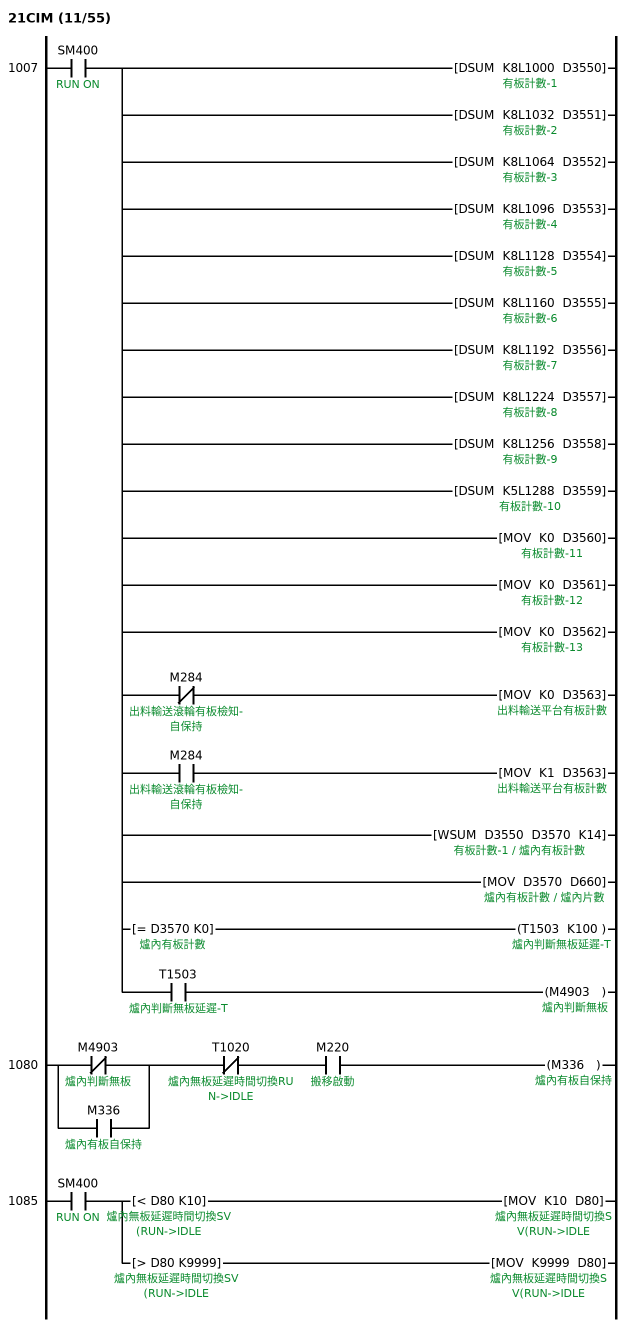
[picture p120: ladder of 21CIM, rungs at steps 1007 to 1085]
1007  LD      SM400  ; RUN ON
      DSUM    K8L1000 D3550  ; 上板記憶 / 有板計數-1
      DSUM    K8L1032 D3551  ; 上板記憶 / 有板計數-2
      DSUM    K8L1064 D3552  ; 上板記憶 / 有板計數-3
      DSUM    K8L1096 D3553  ; 上板記憶 / 有板計數-4
      DSUM    K8L1128 D3554  ; 上板記憶 / 有板計數-5
      DSUM    K8L1160 D3555  ; 上板記憶 / 有板計數-6
      DSUM    K8L1192 D3556  ; 上板記憶 / 有板計數-7
      DSUM    K8L1224 D3557  ; 上板記憶 / 有板計數-8
      DSUM    K8L1256 D3558  ; 上板記憶 / 有板計數-9
      DSUM    K5L1288 D3559  ; 上板記憶 / 有板計數-10
      MOV     K0 D3560  ; 有板計數-11
      MOV     K0 D3561  ; 有板計數-12
      MOV     K0 D3562  ; 有板計數-13
      MPS
      ANI     M284  ; 出料輸送滾輪有板檢知-自保持
      MOV     K0 D3563  ; 出料輸送平台有板計數
      MRD
      AND     M284  ; 出料輸送滾輪有板檢知-自保持
      MOV     K1 D3563
      MPP
      WSUM    D3550 D3570 K14  ; 爐內有板計數
      MOV     D3570 D660  ; 爐內片數
      MPS
      AND=    D3570 K0  ; 爐內有板計數
      OUT     T1503 K100  ; 爐內判斷無板延遲-T
      MPP
      AND     T1503  ; 爐內判斷無板延遲-T
      OUT     M4903  ; 爐內判斷無板
1080  LDI     M4903  ; 爐內判斷無板
      OR      M336  ; 爐內有板自保持
      ANI     T1020  ; 爐內無板延遲時間切換RUN->IDLE
      AND     M220  ; 搬移啟動
      OUT     M336  ; 爐內有板自保持
1085  LD      SM400  ; RUN ON
      MPS
      AND<    D80 K10  ; 爐內無板延遲時間切換SV(RUN->IDLE
      MOV     K10 D80
      MPP
      AND>    D80 K9999  ; 爐內無板延遲時間切換SV(RUN->IDLE
      MOV     K9999 D80
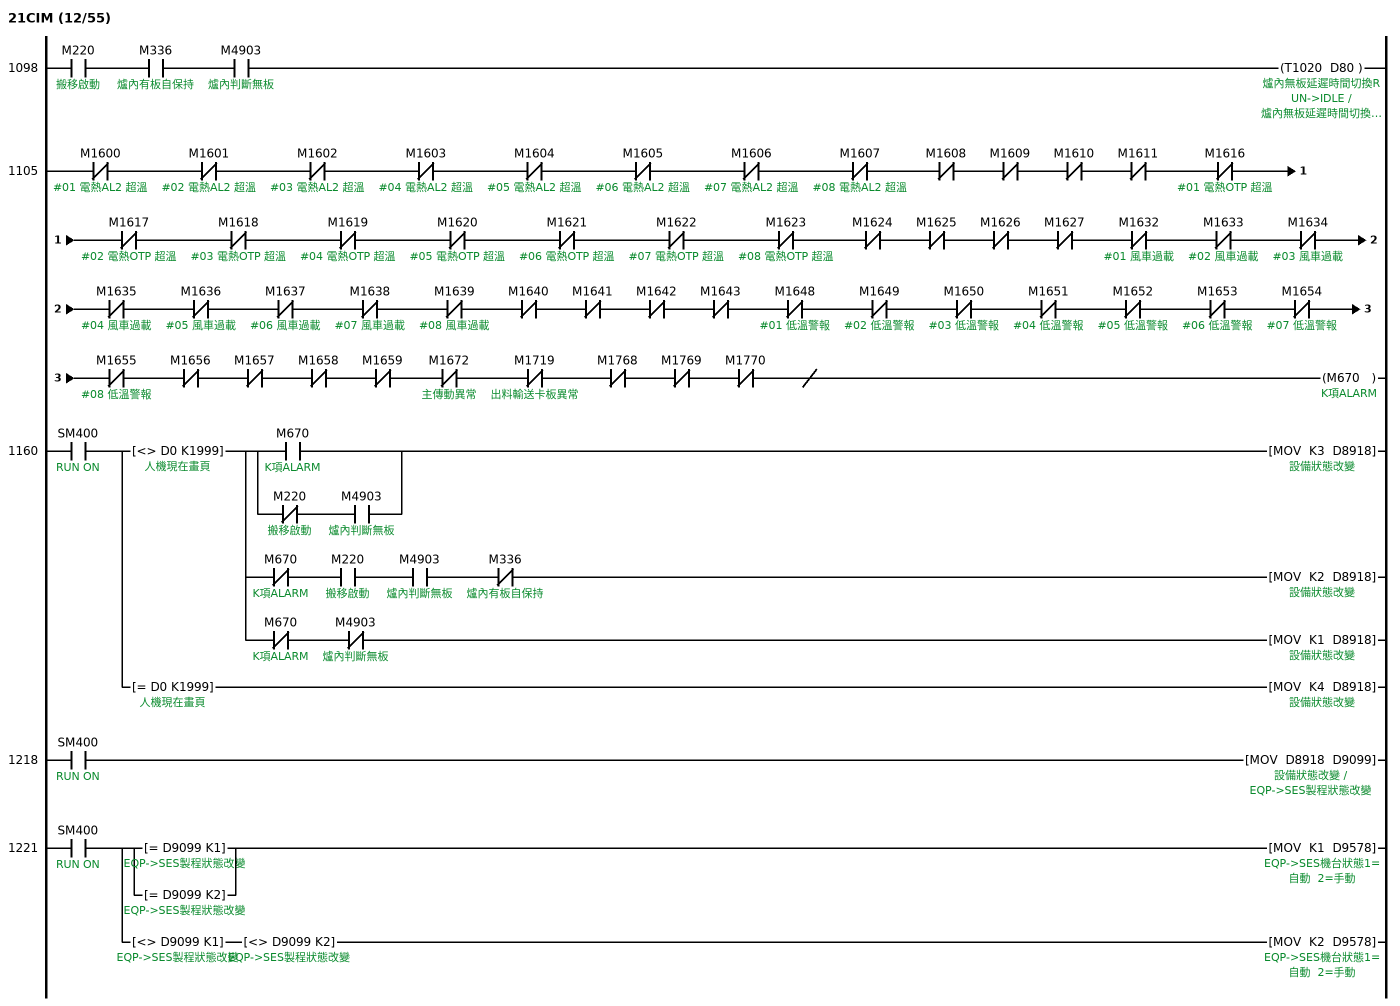
1098  LD      M220  ; 搬移啟動
      AND     M336  ; 爐內有板自保持
      AND     M4903  ; 爐內判斷無板
      OUT     T1020 D80  ; 爐內無板延遲時間切換RUN->IDLE / 爐內無板延遲時間切換SV(RUN->IDLE
1105  LDI     M1600  ; #01 電熱AL2 超溫
      ANI     M1601  ; #02 電熱AL2 超溫
      ANI     M1602  ; #03 電熱AL2 超溫
      ANI     M1603  ; #04 電熱AL2 超溫
      ANI     M1604  ; #05 電熱AL2 超溫
      ANI     M1605  ; #06 電熱AL2 超溫
      ANI     M1606  ; #07 電熱AL2 超溫
      ANI     M1607  ; #08 電熱AL2 超溫
      ANI     M1608
      ANI     M1609
      ANI     M1610
      ANI     M1611
      ANI     M1616  ; #01 電熱OTP 超溫
      ANI     M1617  ; #02 電熱OTP 超溫
      ANI     M1618  ; #03 電熱OTP 超溫
      ANI     M1619  ; #04 電熱OTP 超溫
      ANI     M1620  ; #05 電熱OTP 超溫
      ANI     M1621  ; #06 電熱OTP 超溫
      ANI     M1622  ; #07 電熱OTP 超溫
      ANI     M1623  ; #08 電熱OTP 超溫
      ANI     M1624
      ANI     M1625
      ANI     M1626
      ANI     M1627
      ANI     M1632  ; #01 風車過載
      ANI     M1633  ; #02 風車過載
      ANI     M1634  ; #03 風車過載
      ANI     M1635  ; #04 風車過載
      ANI     M1636  ; #05 風車過載
      ANI     M1637  ; #06 風車過載
      ANI     M1638  ; #07 風車過載
      ANI     M1639  ; #08 風車過載
      ANI     M1640
      ANI     M1641
      ANI     M1642
      ANI     M1643
      ANI     M1648  ; #01 低溫警報
      ANI     M1649  ; #02 低溫警報
      ANI     M1650  ; #03 低溫警報
      ANI     M1651  ; #04 低溫警報
      ANI     M1652  ; #05 低溫警報
      ANI     M1653  ; #06 低溫警報
      ANI     M1654  ; #07 低溫警報
      ANI     M1655  ; #08 低溫警報
      ANI     M1656
      ANI     M1657
      ANI     M1658
      ANI     M1659
      ANI     M1672  ; 主傳動異常
      ANI     M1719  ; 出料輸送卡板異常
      ANI     M1768
      ANI     M1769
      ANI     M1770
      INV
      OUT     M670  ; K項ALARM
1160  LD      SM400  ; RUN ON
      MPS
      AND<>   D0 K1999  ; 人機現在畫頁
      MPS
      LD      M670  ; K項ALARM
      LDI     M220  ; 搬移啟動
      AND     M4903  ; 爐內判斷無板
      ORB
      ANB
      MOV     K3 D8918  ; 設備狀態改變
        [note] State=DOWN
      MRD
      ANI     M670  ; K項ALARM
      AND     M220  ; 搬移啟動
      AND     M4903  ; 爐內判斷無板
      ANI     M336  ; 爐內有板自保持
      MOV     K2 D8918
        [note] State=IDLE
      MPP
      ANI     M670  ; K項ALARM
      ANI     M4903  ; 爐內判斷無板
      MOV     K1 D8918
        [note] State=RUN
      MPP
      AND=    D0 K1999  ; 人機現在畫頁
      MOV     K4 D8918
        [note] State=PM
1218  LD      SM400  ; RUN ON
      MOV     D8918 D9099  ; EQP->SES製程狀態改變
1221  LD      SM400  ; RUN ON
      MPS
      LD=     D9099 K1  ; EQP->SES製程狀態改變
      OR=     D9099 K2  ; EQP->SES製程狀態改變
      ANB
      MOV     K1 D9578  ; EQP->SES機台狀態1=自動  2=手動
      MPP
      AND<>   D9099 K1  ; EQP->SES製程狀態改變
      AND<>   D9099 K2  ; EQP->SES製程狀態改變
      MOV     K2 D9578
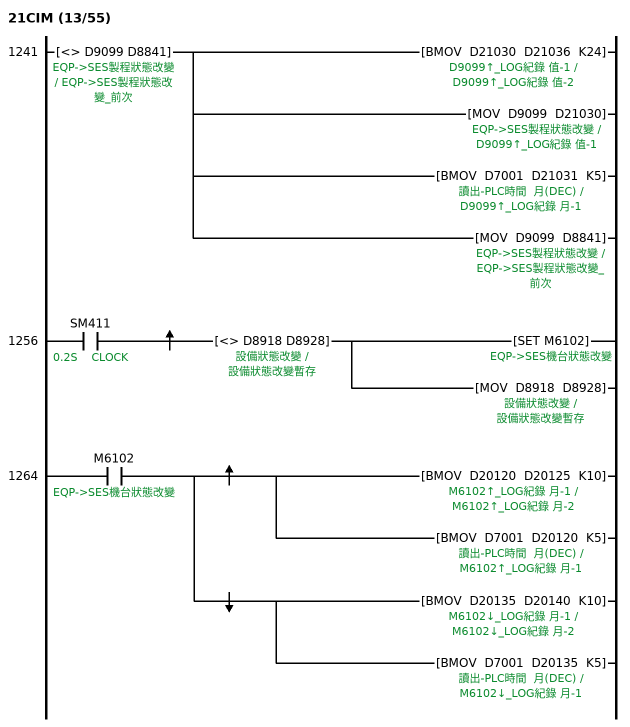
1241  LD<>    D9099 D8841  ; EQP->SES製程狀態改變 / EQP->SES製程狀態改變_前次
      BMOV    D21030 D21036 K24  ; D9099↑_LOG紀錄 值-1 / D9099↑_LOG紀錄 值-2
      MOV     D9099 D21030
      BMOV    D7001 D21031 K5  ; D9099↑_LOG紀錄 月-1
      MOV     D9099 D8841
1256  LD      SM411  ; 0.2S    CLOCK
      MEP
      AND<>   D8918 D8928  ; 設備狀態改變 / 設備狀態改變暫存
      SET     M6102  ; EQP->SES機台狀態改變
      MOV     D8918 D8928
1264  LD      M6102  ; EQP->SES機台狀態改變
      MPS
      MEP
      BMOV    D20120 D20125 K10  ; M6102↑_LOG紀錄 月-1 / M6102↑_LOG紀錄 月-2
      BMOV    D7001 D20120 K5
      MPP
      MEF
      BMOV    D20135 D20140 K10  ; M6102↓_LOG紀錄 月-1 / M6102↓_LOG紀錄 月-2
      BMOV    D7001 D20135 K5
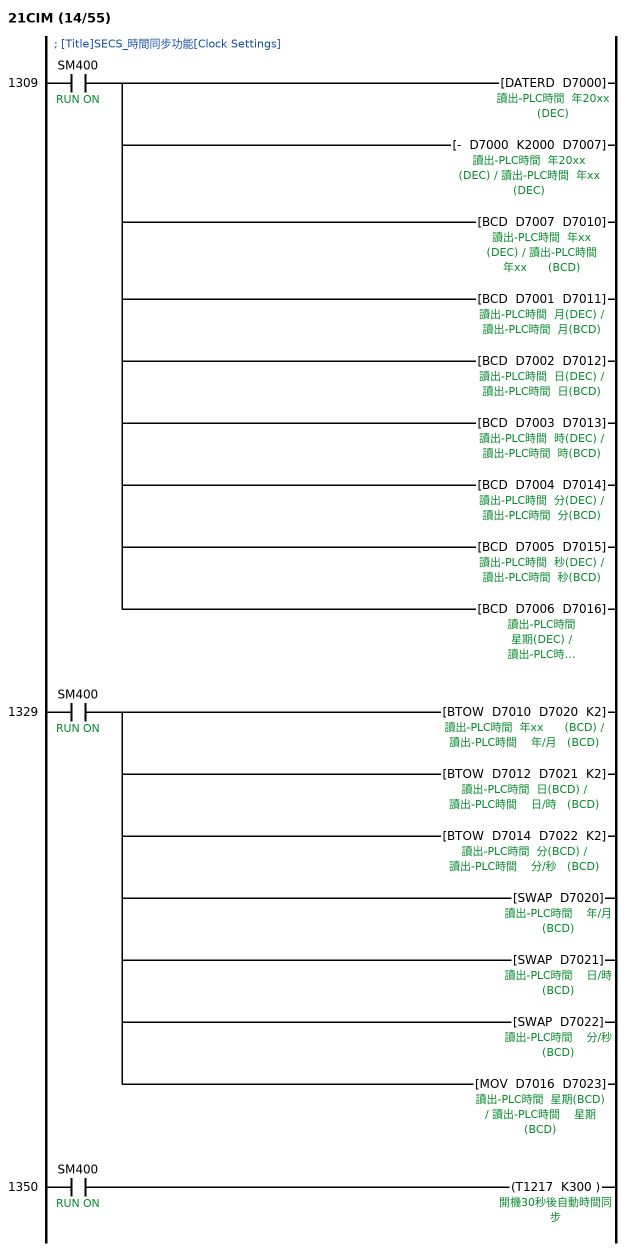
; [Title]SECS_時間同步功能[Clock Settings]
1309  LD      SM400  ; RUN ON
      DATERD  D7000  ; 讀出-PLC時間  年20xx    (DEC)
      -       D7000 K2000 D7007  ; 讀出-PLC時間  年xx      (DEC)
      BCD     D7007 D7010  ; 讀出-PLC時間  年xx      (BCD)
      BCD     D7001 D7011  ; 讀出-PLC時間  月(BCD)
      BCD     D7002 D7012  ; 讀出-PLC時間  日(DEC) / 讀出-PLC時間  日(BCD)
      BCD     D7003 D7013  ; 讀出-PLC時間  時(DEC) / 讀出-PLC時間  時(BCD)
      BCD     D7004 D7014  ; 讀出-PLC時間  分(DEC) / 讀出-PLC時間  分(BCD)
      BCD     D7005 D7015  ; 讀出-PLC時間  秒(DEC) / 讀出-PLC時間  秒(BCD)
      BCD     D7006 D7016  ; 讀出-PLC時間  星期(DEC) / 讀出-PLC時間  星期(BCD)
1329  LD      SM400  ; RUN ON
      BTOW    D7010 D7020 K2  ; 讀出-PLC時間    年/月   (BCD)
      BTOW    D7012 D7021 K2  ; 讀出-PLC時間    日/時   (BCD)
      BTOW    D7014 D7022 K2  ; 讀出-PLC時間    分/秒   (BCD)
      SWAP    D7020
      SWAP    D7021
      SWAP    D7022
      MOV     D7016 D7023  ; 讀出-PLC時間    星期    (BCD)
1350  LD      SM400  ; RUN ON
      OUT     T1217 K300  ; 開機30秒後自動時間同步
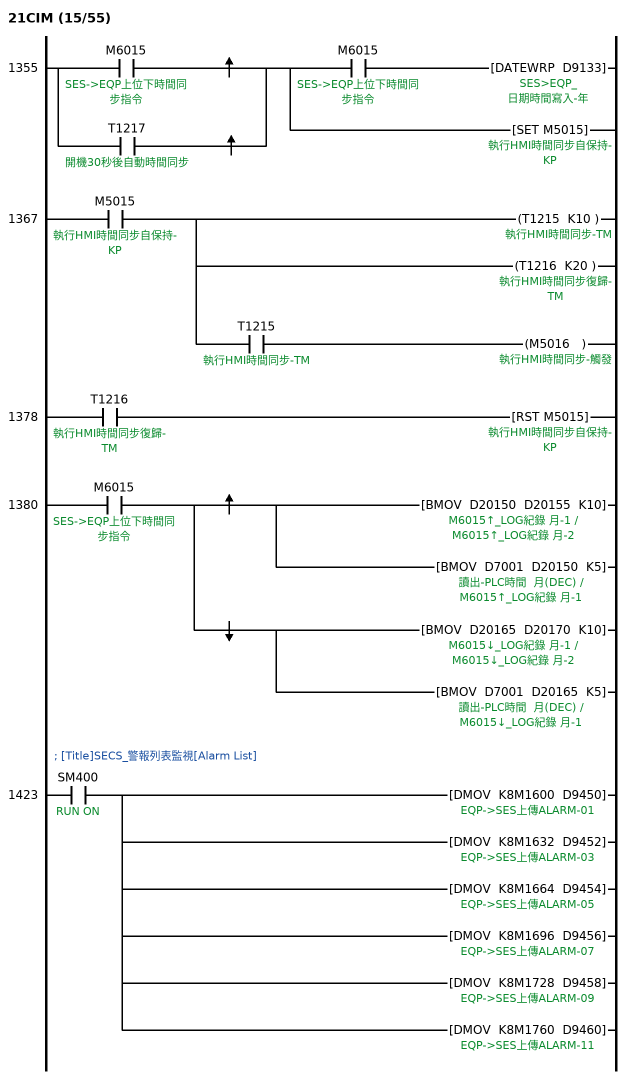
1355  LD      M6015  ; SES->EQP上位下時間同步指令
      MEP
      LD      T1217  ; 開機30秒後自動時間同步
      MEP
      ORB
      MPS
      AND     M6015  ; SES->EQP上位下時間同步指令
      DATEWRP D9133  ; SES>EQP_日期時間寫入-年
      MPP
      SET     M5015  ; 執行HMI時間同步自保持-KP
1367  LD      M5015  ; 執行HMI時間同步自保持-KP
      OUT     T1215 K10  ; 執行HMI時間同步-TM
      OUT     T1216 K20  ; 執行HMI時間同步復歸-TM
      AND     T1215  ; 執行HMI時間同步-TM
      OUT     M5016  ; 執行HMI時間同步-觸發
1378  LD      T1216  ; 執行HMI時間同步復歸-TM
      RST     M5015  ; 執行HMI時間同步自保持-KP
1380  LD      M6015  ; SES->EQP上位下時間同步指令
      MPS
      MEP
      BMOV    D20150 D20155 K10  ; M6015↑_LOG紀錄 月-1 / M6015↑_LOG紀錄 月-2
      BMOV    D7001 D20150 K5
      MPP
      MEF
      BMOV    D20165 D20170 K10  ; M6015↓_LOG紀錄 月-1 / M6015↓_LOG紀錄 月-2
      BMOV    D7001 D20165 K5
; [Title]SECS_警報列表監視[Alarm List]
1423  LD      SM400  ; RUN ON
      DMOV    K8M1600 D9450  ; EQP->SES上傳ALARM-01
      DMOV    K8M1632 D9452  ; EQP->SES上傳ALARM-03
      DMOV    K8M1664 D9454  ; EQP->SES上傳ALARM-05
      DMOV    K8M1696 D9456  ; EQP->SES上傳ALARM-07
      DMOV    K8M1728 D9458  ; EQP->SES上傳ALARM-09
      DMOV    K8M1760 D9460  ; EQP->SES上傳ALARM-11
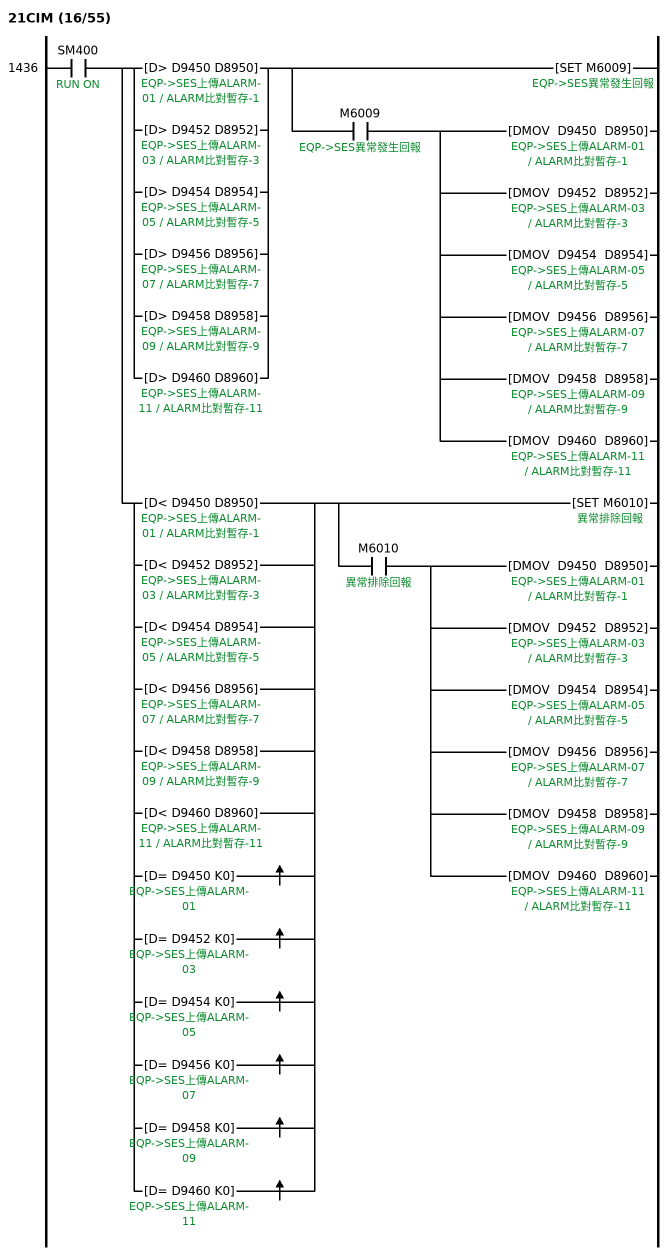
1436  LD      SM400  ; RUN ON
      MPS
      LDD>    D9450 D8950  ; EQP->SES上傳ALARM-01 / ALARM比對暫存-1
      ORD>    D9452 D8952  ; EQP->SES上傳ALARM-03 / ALARM比對暫存-3
      ORD>    D9454 D8954  ; EQP->SES上傳ALARM-05 / ALARM比對暫存-5
      ORD>    D9456 D8956  ; EQP->SES上傳ALARM-07 / ALARM比對暫存-7
      ORD>    D9458 D8958  ; EQP->SES上傳ALARM-09 / ALARM比對暫存-9
      ORD>    D9460 D8960  ; EQP->SES上傳ALARM-11 / ALARM比對暫存-11
      ANB
      SET     M6009  ; EQP->SES異常發生回報
      AND     M6009  ; EQP->SES異常發生回報
      DMOV    D9450 D8950
      DMOV    D9452 D8952
      DMOV    D9454 D8954
      DMOV    D9456 D8956
      DMOV    D9458 D8958
      DMOV    D9460 D8960
      MPP
      LDD<    D9450 D8950  ; EQP->SES上傳ALARM-01 / ALARM比對暫存-1
      ORD<    D9452 D8952  ; EQP->SES上傳ALARM-03 / ALARM比對暫存-3
      ORD<    D9454 D8954  ; EQP->SES上傳ALARM-05 / ALARM比對暫存-5
      ORD<    D9456 D8956  ; EQP->SES上傳ALARM-07 / ALARM比對暫存-7
      ORD<    D9458 D8958  ; EQP->SES上傳ALARM-09 / ALARM比對暫存-9
      ORD<    D9460 D8960  ; EQP->SES上傳ALARM-11 / ALARM比對暫存-11
      LDD=    D9450 K0  ; EQP->SES上傳ALARM-01
      MEP
      ORB
      LDD=    D9452 K0  ; EQP->SES上傳ALARM-03
      MEP
      ORB
      LDD=    D9454 K0  ; EQP->SES上傳ALARM-05
      MEP
      ORB
      LDD=    D9456 K0  ; EQP->SES上傳ALARM-07
      MEP
      ORB
      LDD=    D9458 K0  ; EQP->SES上傳ALARM-09
      MEP
      ORB
      LDD=    D9460 K0  ; EQP->SES上傳ALARM-11
      MEP
      ORB
      ANB
      SET     M6010  ; 異常排除回報
      AND     M6010  ; 異常排除回報
      DMOV    D9450 D8950
      DMOV    D9452 D8952
      DMOV    D9454 D8954
      DMOV    D9456 D8956
      DMOV    D9458 D8958
      DMOV    D9460 D8960
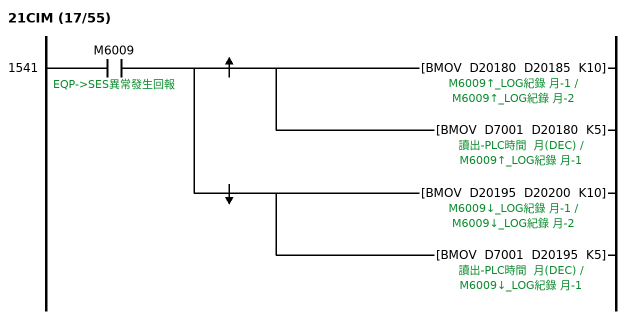
1541  LD      M6009  ; EQP->SES異常發生回報
      MPS
      MEP
      BMOV    D20180 D20185 K10  ; M6009↑_LOG紀錄 月-1 / M6009↑_LOG紀錄 月-2
      BMOV    D7001 D20180 K5
      MPP
      MEF
      BMOV    D20195 D20200 K10  ; M6009↓_LOG紀錄 月-1 / M6009↓_LOG紀錄 月-2
      BMOV    D7001 D20195 K5
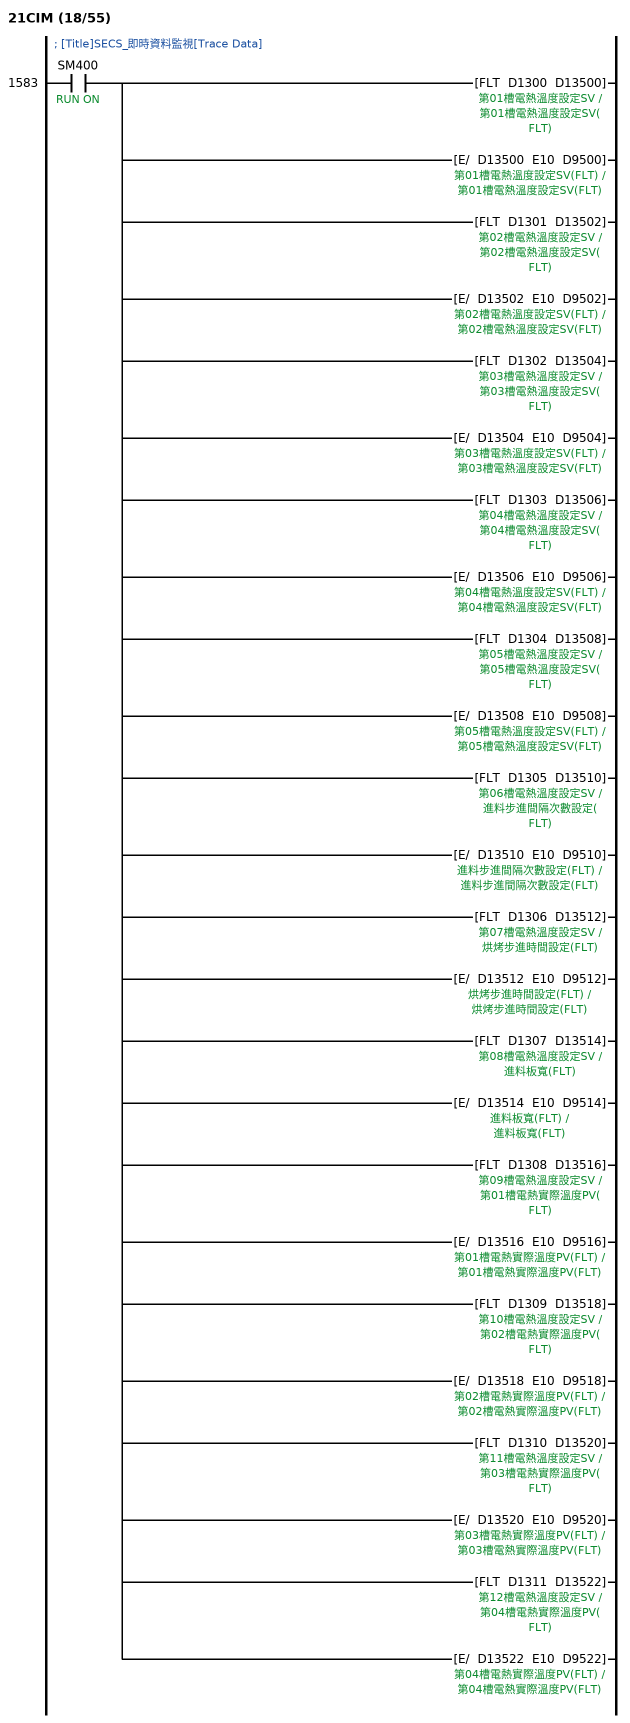
; [Title]SECS_即時資料監視[Trace Data]
1583  LD      SM400  ; RUN ON
      FLT     D1300 D13500  ; 第01槽電熱溫度設定SV(FLT)
      E/      D13500 E10 D9500  ; 第01槽電熱溫度設定SV(FLT)
      FLT     D1301 D13502  ; 第02槽電熱溫度設定SV / 第02槽電熱溫度設定SV(FLT)
      E/      D13502 E10 D9502  ; 第02槽電熱溫度設定SV(FLT)
      FLT     D1302 D13504  ; 第03槽電熱溫度設定SV / 第03槽電熱溫度設定SV(FLT)
      E/      D13504 E10 D9504  ; 第03槽電熱溫度設定SV(FLT)
      FLT     D1303 D13506  ; 第04槽電熱溫度設定SV / 第04槽電熱溫度設定SV(FLT)
      E/      D13506 E10 D9506  ; 第04槽電熱溫度設定SV(FLT)
      FLT     D1304 D13508  ; 第05槽電熱溫度設定SV / 第05槽電熱溫度設定SV(FLT)
      E/      D13508 E10 D9508  ; 第05槽電熱溫度設定SV(FLT)
      FLT     D1305 D13510  ; 第06槽電熱溫度設定SV / 進料步進間隔次數設定(FLT)
      E/      D13510 E10 D9510  ; 進料步進間隔次數設定(FLT)
      FLT     D1306 D13512  ; 第07槽電熱溫度設定SV / 烘烤步進時間設定(FLT)
      E/      D13512 E10 D9512  ; 烘烤步進時間設定(FLT)
      FLT     D1307 D13514  ; 第08槽電熱溫度設定SV / 進料板寬(FLT)
      E/      D13514 E10 D9514  ; 進料板寬(FLT)
      FLT     D1308 D13516  ; 第09槽電熱溫度設定SV / 第01槽電熱實際溫度PV(FLT)
      E/      D13516 E10 D9516  ; 第01槽電熱實際溫度PV(FLT)
      FLT     D1309 D13518  ; 第10槽電熱溫度設定SV / 第02槽電熱實際溫度PV(FLT)
      E/      D13518 E10 D9518  ; 第02槽電熱實際溫度PV(FLT)
      FLT     D1310 D13520  ; 第11槽電熱溫度設定SV / 第03槽電熱實際溫度PV(FLT)
      E/      D13520 E10 D9520  ; 第03槽電熱實際溫度PV(FLT)
      FLT     D1311 D13522  ; 第12槽電熱溫度設定SV / 第04槽電熱實際溫度PV(FLT)
      E/      D13522 E10 D9522  ; 第04槽電熱實際溫度PV(FLT)
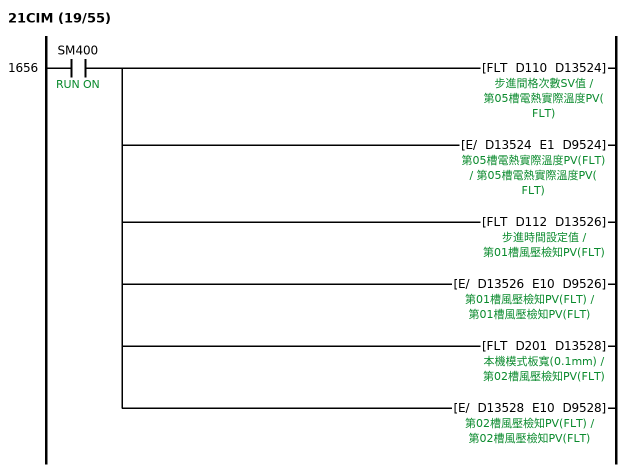
1656  LD      SM400  ; RUN ON
      FLT     D110 D13524  ; 第05槽電熱實際溫度PV(FLT)
      E/      D13524 E1 D9524  ; 第05槽電熱實際溫度PV(FLT)
      FLT     D112 D13526  ; 第01槽風壓檢知PV(FLT)
      E/      D13526 E10 D9526  ; 第01槽風壓檢知PV(FLT)
      FLT     D201 D13528  ; 第02槽風壓檢知PV(FLT)
      E/      D13528 E10 D9528  ; 第02槽風壓檢知PV(FLT)
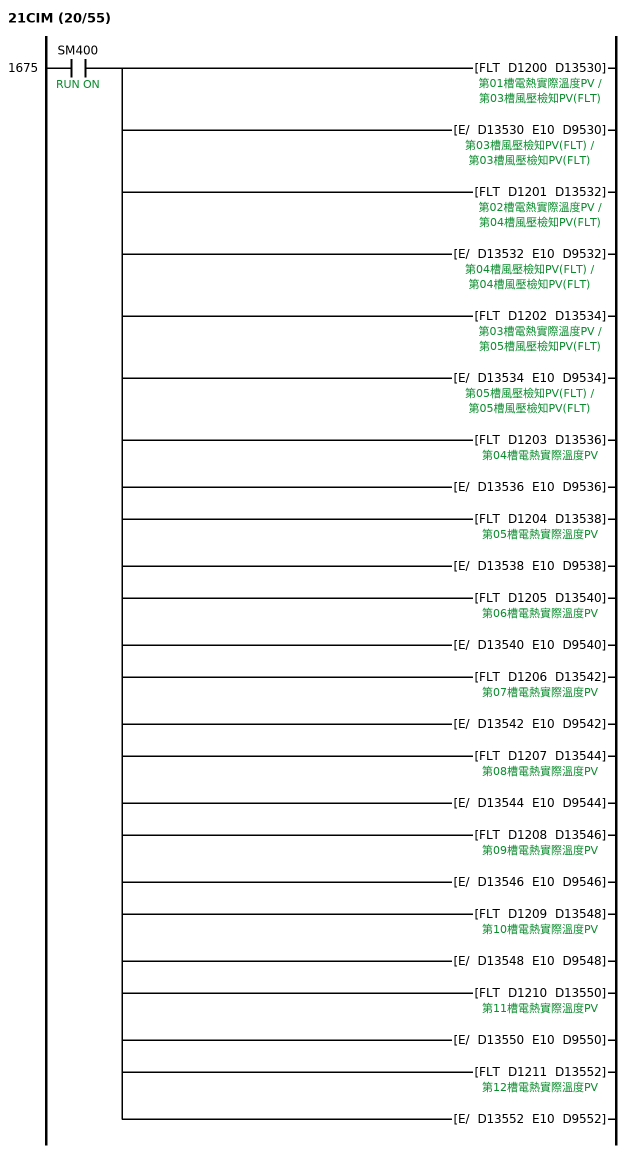
1675  LD      SM400  ; RUN ON
      FLT     D1200 D13530  ; 第03槽風壓檢知PV(FLT)
      E/      D13530 E10 D9530  ; 第03槽風壓檢知PV(FLT)
      FLT     D1201 D13532  ; 第02槽電熱實際溫度PV / 第04槽風壓檢知PV(FLT)
      E/      D13532 E10 D9532  ; 第04槽風壓檢知PV(FLT)
      FLT     D1202 D13534  ; 第03槽電熱實際溫度PV / 第05槽風壓檢知PV(FLT)
      E/      D13534 E10 D9534  ; 第05槽風壓檢知PV(FLT)
      FLT     D1203 D13536  ; 第04槽電熱實際溫度PV
      E/      D13536 E10 D9536
      FLT     D1204 D13538  ; 第05槽電熱實際溫度PV
      E/      D13538 E10 D9538
      FLT     D1205 D13540  ; 第06槽電熱實際溫度PV
      E/      D13540 E10 D9540
      FLT     D1206 D13542  ; 第07槽電熱實際溫度PV
      E/      D13542 E10 D9542
      FLT     D1207 D13544  ; 第08槽電熱實際溫度PV
      E/      D13544 E10 D9544
      FLT     D1208 D13546  ; 第09槽電熱實際溫度PV
      E/      D13546 E10 D9546
      FLT     D1209 D13548  ; 第10槽電熱實際溫度PV
      E/      D13548 E10 D9548
      FLT     D1210 D13550  ; 第11槽電熱實際溫度PV
      E/      D13550 E10 D9550
      FLT     D1211 D13552
      E/      D13552 E10 D9552
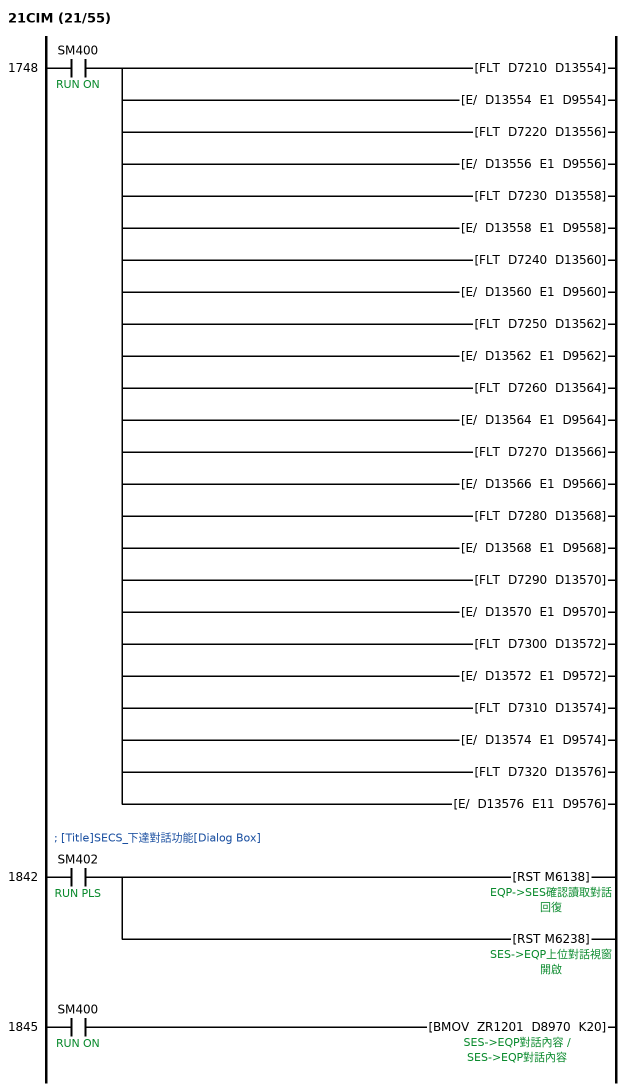
1748  LD      SM400  ; RUN ON
      FLT     D7210 D13554
      E/      D13554 E1 D9554
      FLT     D7220 D13556
      E/      D13556 E1 D9556
      FLT     D7230 D13558
      E/      D13558 E1 D9558
      FLT     D7240 D13560
      E/      D13560 E1 D9560
      FLT     D7250 D13562
      E/      D13562 E1 D9562
      FLT     D7260 D13564
      E/      D13564 E1 D9564
      FLT     D7270 D13566
      E/      D13566 E1 D9566
      FLT     D7280 D13568
      E/      D13568 E1 D9568
      FLT     D7290 D13570
      E/      D13570 E1 D9570
      FLT     D7300 D13572
      E/      D13572 E1 D9572
      FLT     D7310 D13574
      E/      D13574 E1 D9574
      FLT     D7320 D13576
      E/      D13576 E11 D9576
; [Title]SECS_下達對話功能[Dialog Box]
1842  LD      SM402  ; RUN PLS
      RST     M6138  ; EQP->SES確認讀取對話回復
      RST     M6238  ; SES->EQP上位對話視窗開啟
1845  LD      SM400  ; RUN ON
      BMOV    ZR1201 D8970 K20  ; SES->EQP對話內容 / SES->EQP對話內容
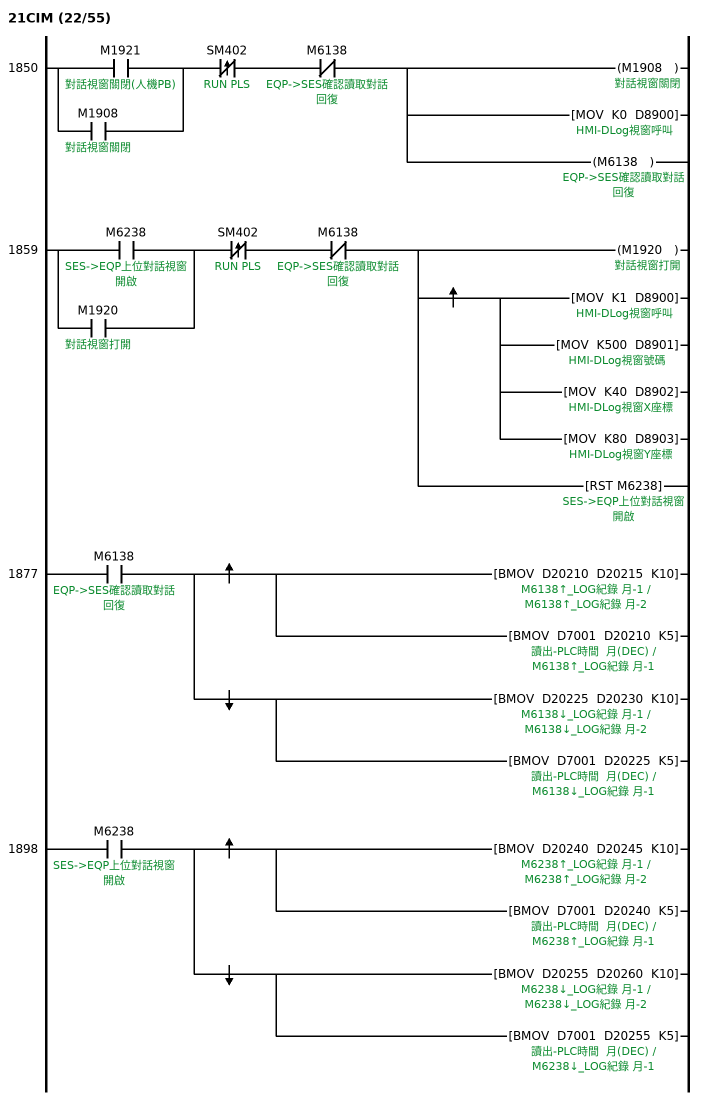
1850  LD      M1921  ; 對話視窗關閉(人機PB)
      OR      M1908  ; 對話視窗關閉
      ANDPI   SM402  ; RUN PLS
      ANI     M6138  ; EQP->SES確認讀取對話回復
      OUT     M1908  ; 對話視窗關閉
      MOV     K0 D8900  ; HMI-DLog視窗呼叫
      OUT     M6138  ; EQP->SES確認讀取對話回復
1859  LD      M6238  ; SES->EQP上位對話視窗開啟
      OR      M1920  ; 對話視窗打開
      ANDPI   SM402  ; RUN PLS
      ANI     M6138  ; EQP->SES確認讀取對話回復
      OUT     M1920  ; 對話視窗打開
      MPS
      MEP
      MOV     K1 D8900
      MOV     K500 D8901  ; HMI-DLog視窗號碼
      MOV     K40 D8902  ; HMI-DLog視窗X座標
      MOV     K80 D8903  ; HMI-DLog視窗Y座標
      MPP
      RST     M6238  ; SES->EQP上位對話視窗開啟
1877  LD      M6138  ; EQP->SES確認讀取對話回復
      MPS
      MEP
      BMOV    D20210 D20215 K10  ; M6138↑_LOG紀錄 月-1 / M6138↑_LOG紀錄 月-2
      BMOV    D7001 D20210 K5
      MPP
      MEF
      BMOV    D20225 D20230 K10  ; M6138↓_LOG紀錄 月-1 / M6138↓_LOG紀錄 月-2
      BMOV    D7001 D20225 K5
1898  LD      M6238  ; SES->EQP上位對話視窗開啟
      MPS
      MEP
      BMOV    D20240 D20245 K10  ; M6238↑_LOG紀錄 月-1 / M6238↑_LOG紀錄 月-2
      BMOV    D7001 D20240 K5
      MPP
      MEF
      BMOV    D20255 D20260 K10  ; M6238↓_LOG紀錄 月-1 / M6238↓_LOG紀錄 月-2
      BMOV    D7001 D20255 K5
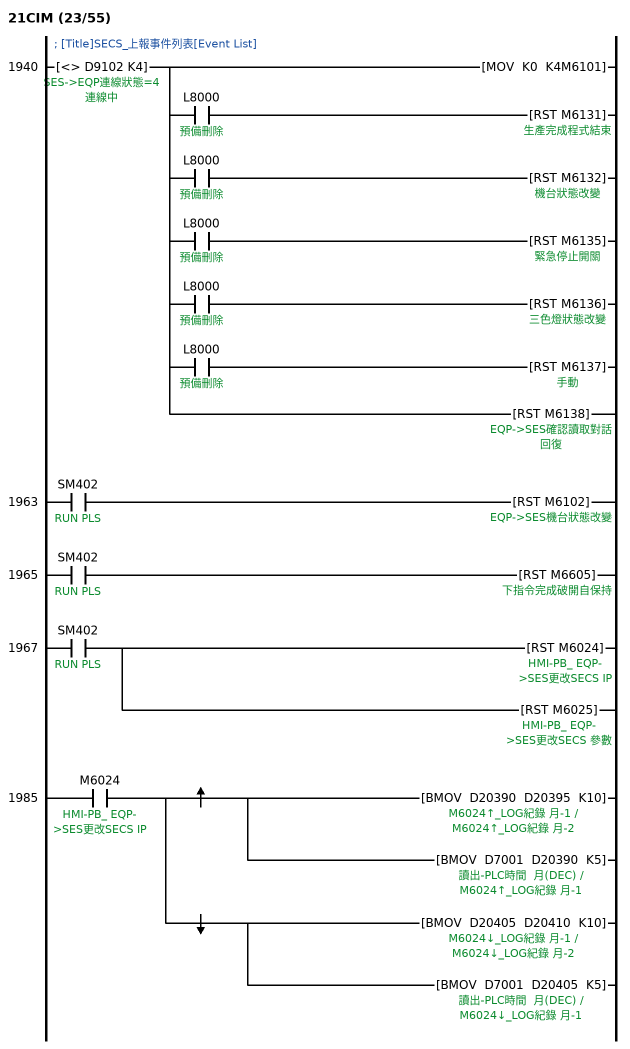
; [Title]SECS_上報事件列表[Event List]
1940  LD<>    D9102 K4  ; SES->EQP連線狀態=4      連線中
      MOV     K0 K4M6101
      MPS
      AND     L8000  ; 預備刪除
      RST     M6131  ; 生產完成程式結束
      MRD
      AND     L8000  ; 預備刪除
      RST     M6132  ; 機台狀態改變
      MRD
      AND     L8000  ; 預備刪除
      RST     M6135  ; 緊急停止開關
      MRD
      AND     L8000  ; 預備刪除
      RST     M6136  ; 三色燈狀態改變
      MRD
      AND     L8000  ; 預備刪除
      RST     M6137  ; 手動
      MPP
      RST     M6138  ; EQP->SES確認讀取對話回復
1963  LD      SM402  ; RUN PLS
      RST     M6102  ; EQP->SES機台狀態改變
1965  LD      SM402  ; RUN PLS
      RST     M6605  ; 下指令完成破開自保持
1967  LD      SM402  ; RUN PLS
      RST     M6024  ; HMI-PB_ EQP->SES更改SECS IP
        [note] HMI上變更C語言模組網路設定
      RST     M6025  ; HMI-PB_ EQP->SES更改SECS 參數
1985  LD      M6024  ; HMI-PB_ EQP->SES更改SECS IP
      MPS
      MEP
      BMOV    D20390 D20395 K10  ; M6024↑_LOG紀錄 月-1 / M6024↑_LOG紀錄 月-2
      BMOV    D7001 D20390 K5
      MPP
      MEF
      BMOV    D20405 D20410 K10  ; M6024↓_LOG紀錄 月-1 / M6024↓_LOG紀錄 月-2
      BMOV    D7001 D20405 K5
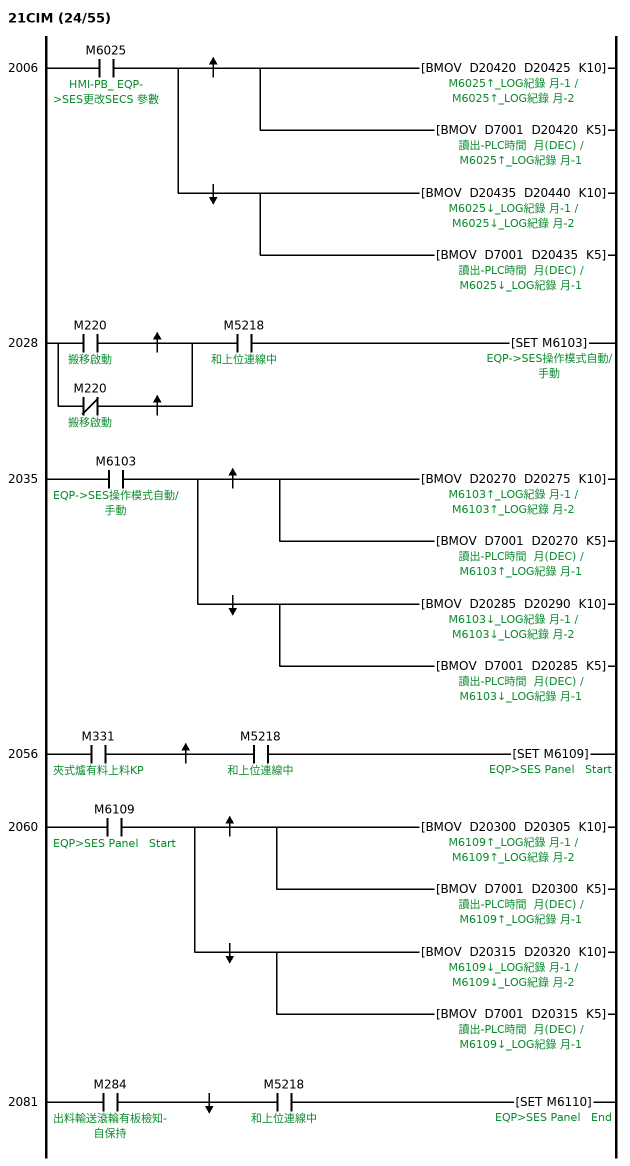
2006  LD      M6025  ; HMI-PB_ EQP->SES更改SECS 參數
      MPS
      MEP
      BMOV    D20420 D20425 K10  ; M6025↑_LOG紀錄 月-1 / M6025↑_LOG紀錄 月-2
      BMOV    D7001 D20420 K5
      MPP
      MEF
      BMOV    D20435 D20440 K10  ; M6025↓_LOG紀錄 月-1 / M6025↓_LOG紀錄 月-2
      BMOV    D7001 D20435 K5
2028  LD      M220  ; 搬移啟動
      MEP
      LDI     M220  ; 搬移啟動
      MEP
      ORB
      AND     M5218  ; 和上位連線中
      SET     M6103  ; EQP->SES操作模式自動/手動
2035  LD      M6103  ; EQP->SES操作模式自動/手動
      MPS
      MEP
      BMOV    D20270 D20275 K10  ; M6103↑_LOG紀錄 月-1 / M6103↑_LOG紀錄 月-2
      BMOV    D7001 D20270 K5
      MPP
      MEF
      BMOV    D20285 D20290 K10  ; M6103↓_LOG紀錄 月-1 / M6103↓_LOG紀錄 月-2
      BMOV    D7001 D20285 K5
2056  LD      M331  ; 夾式爐有料上料KP
      MEP
      AND     M5218  ; 和上位連線中
      SET     M6109  ; EQP>SES Panel   Start
2060  LD      M6109  ; EQP>SES Panel   Start
      MPS
      MEP
      BMOV    D20300 D20305 K10  ; M6109↑_LOG紀錄 月-1 / M6109↑_LOG紀錄 月-2
      BMOV    D7001 D20300 K5
      MPP
      MEF
      BMOV    D20315 D20320 K10  ; M6109↓_LOG紀錄 月-1 / M6109↓_LOG紀錄 月-2
      BMOV    D7001 D20315 K5
2081  LD      M284  ; 出料輸送滾輪有板檢知-自保持
      MEF
      AND     M5218  ; 和上位連線中
      SET     M6110  ; EQP>SES Panel   End
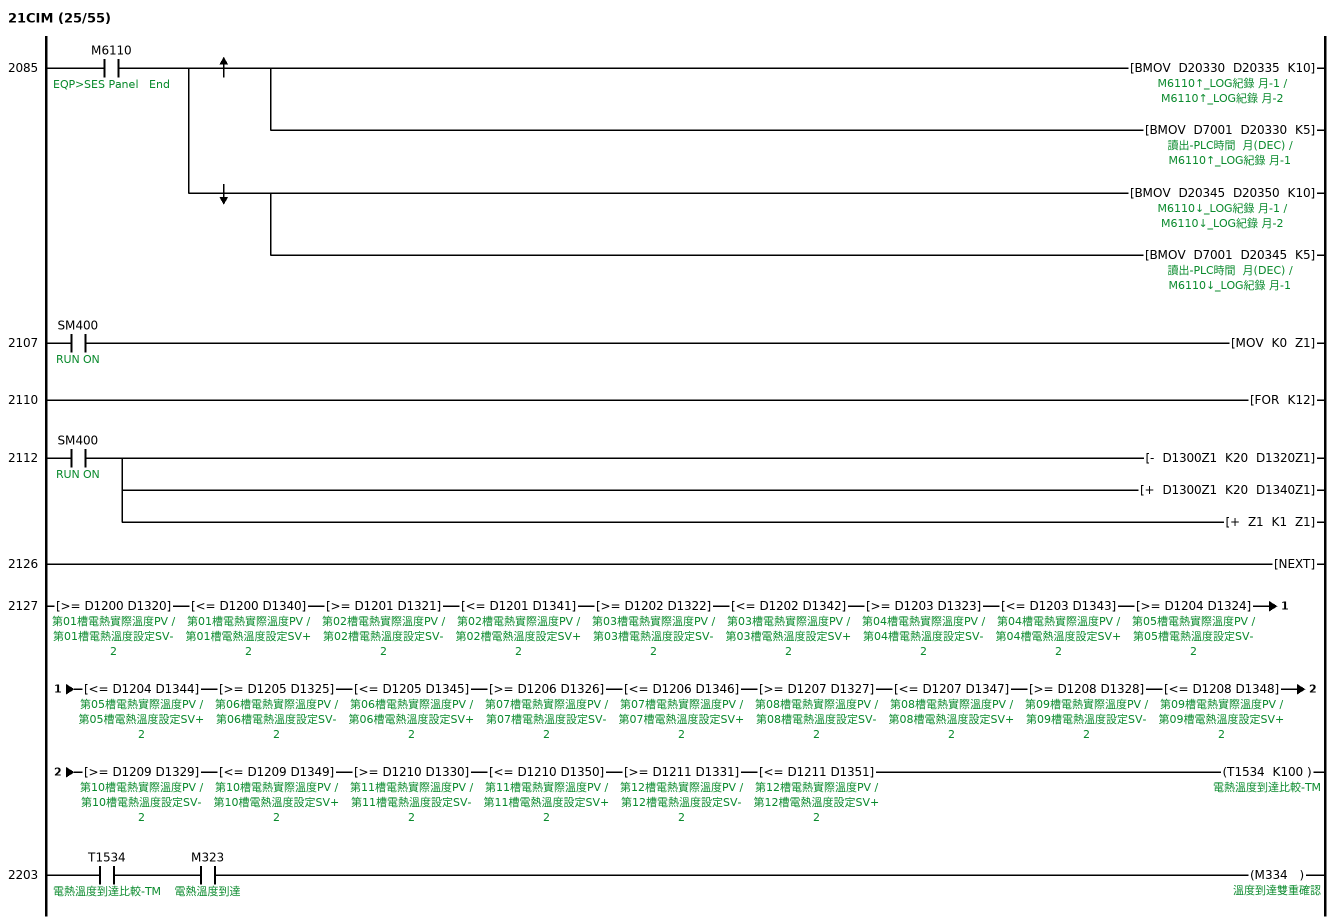
2085  LD      M6110  ; EQP>SES Panel   End
      MPS
      MEP
      BMOV    D20330 D20335 K10  ; M6110↑_LOG紀錄 月-1 / M6110↑_LOG紀錄 月-2
      BMOV    D7001 D20330 K5
      MPP
      MEF
      BMOV    D20345 D20350 K10  ; M6110↓_LOG紀錄 月-1 / M6110↓_LOG紀錄 月-2
      BMOV    D7001 D20345 K5
2107  LD      SM400  ; RUN ON
      MOV     K0 Z1
2110  FOR     K12
2112  LD      SM400  ; RUN ON
      -       D1300Z1 K20 D1320Z1
      +       D1300Z1 K20 D1340Z1
      +       Z1 K1 Z1
2126  NEXT
2127  LD>=    D1200 D1320  ; 第01槽電熱實際溫度PV / 第01槽電熱溫度設定SV-2
      AND<=   D1200 D1340  ; 第01槽電熱實際溫度PV / 第01槽電熱溫度設定SV+2
      AND>=   D1201 D1321  ; 第02槽電熱實際溫度PV / 第02槽電熱溫度設定SV-2
      AND<=   D1201 D1341  ; 第02槽電熱實際溫度PV / 第02槽電熱溫度設定SV+2
      AND>=   D1202 D1322  ; 第03槽電熱實際溫度PV / 第03槽電熱溫度設定SV-2
      AND<=   D1202 D1342  ; 第03槽電熱實際溫度PV / 第03槽電熱溫度設定SV+2
      AND>=   D1203 D1323  ; 第04槽電熱實際溫度PV / 第04槽電熱溫度設定SV-2
      AND<=   D1203 D1343  ; 第04槽電熱實際溫度PV / 第04槽電熱溫度設定SV+2
      AND>=   D1204 D1324  ; 第05槽電熱實際溫度PV / 第05槽電熱溫度設定SV-2
      AND<=   D1204 D1344  ; 第05槽電熱實際溫度PV / 第05槽電熱溫度設定SV+2
      AND>=   D1205 D1325  ; 第06槽電熱實際溫度PV / 第06槽電熱溫度設定SV-2
      AND<=   D1205 D1345  ; 第06槽電熱實際溫度PV / 第06槽電熱溫度設定SV+2
      AND>=   D1206 D1326  ; 第07槽電熱實際溫度PV / 第07槽電熱溫度設定SV-2
      AND<=   D1206 D1346  ; 第07槽電熱實際溫度PV / 第07槽電熱溫度設定SV+2
      AND>=   D1207 D1327  ; 第08槽電熱實際溫度PV / 第08槽電熱溫度設定SV-2
      AND<=   D1207 D1347  ; 第08槽電熱實際溫度PV / 第08槽電熱溫度設定SV+2
      AND>=   D1208 D1328  ; 第09槽電熱實際溫度PV / 第09槽電熱溫度設定SV-2
      AND<=   D1208 D1348  ; 第09槽電熱實際溫度PV / 第09槽電熱溫度設定SV+2
      AND>=   D1209 D1329  ; 第10槽電熱實際溫度PV / 第10槽電熱溫度設定SV-2
      AND<=   D1209 D1349  ; 第10槽電熱實際溫度PV / 第10槽電熱溫度設定SV+2
      AND>=   D1210 D1330  ; 第11槽電熱實際溫度PV / 第11槽電熱溫度設定SV-2
      AND<=   D1210 D1350  ; 第11槽電熱實際溫度PV / 第11槽電熱溫度設定SV+2
      AND>=   D1211 D1331  ; 第12槽電熱實際溫度PV / 第12槽電熱溫度設定SV-2
      AND<=   D1211 D1351  ; 第12槽電熱實際溫度PV / 第12槽電熱溫度設定SV+2
      OUT     T1534 K100  ; 電熱溫度到達比較-TM
2203  LD      T1534  ; 電熱溫度到達比較-TM
      AND     M323  ; 電熱溫度到達
      OUT     M334  ; 溫度到達雙重確認
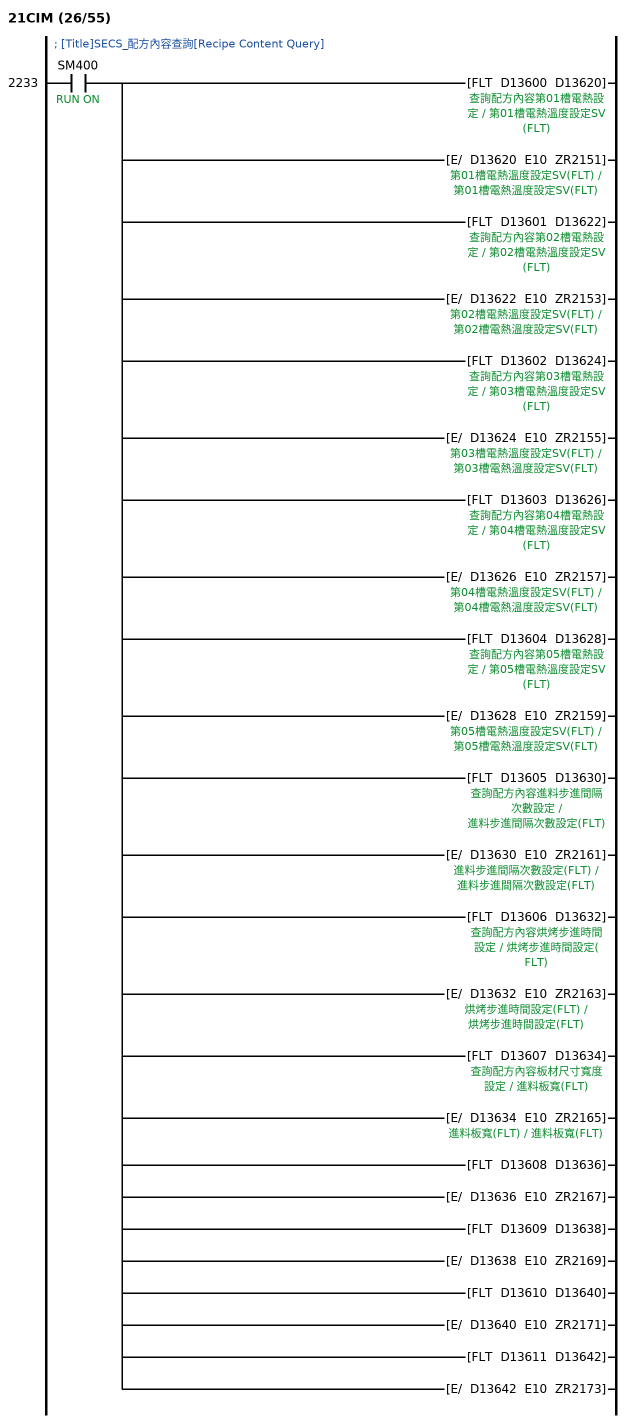
; [Title]SECS_配方內容查詢[Recipe Content Query]
2233  LD      SM400  ; RUN ON
      FLT     D13600 D13620  ; 查詢配方內容第01槽電熱設定 / 第01槽電熱溫度設定SV(FLT)
      E/      D13620 E10 ZR2151  ; 第01槽電熱溫度設定SV(FLT)
      FLT     D13601 D13622  ; 查詢配方內容第02槽電熱設定 / 第02槽電熱溫度設定SV(FLT)
      E/      D13622 E10 ZR2153  ; 第02槽電熱溫度設定SV(FLT)
      FLT     D13602 D13624  ; 查詢配方內容第03槽電熱設定 / 第03槽電熱溫度設定SV(FLT)
      E/      D13624 E10 ZR2155  ; 第03槽電熱溫度設定SV(FLT)
      FLT     D13603 D13626  ; 查詢配方內容第04槽電熱設定 / 第04槽電熱溫度設定SV(FLT)
      E/      D13626 E10 ZR2157  ; 第04槽電熱溫度設定SV(FLT)
      FLT     D13604 D13628  ; 查詢配方內容第05槽電熱設定 / 第05槽電熱溫度設定SV(FLT)
      E/      D13628 E10 ZR2159  ; 第05槽電熱溫度設定SV(FLT)
      FLT     D13605 D13630  ; 查詢配方內容進料步進間隔次數設定 / 進料步進間隔次數設定(FLT)
      E/      D13630 E10 ZR2161  ; 進料步進間隔次數設定(FLT)
      FLT     D13606 D13632  ; 查詢配方內容烘烤步進時間設定 / 烘烤步進時間設定(FLT)
      E/      D13632 E10 ZR2163  ; 烘烤步進時間設定(FLT)
      FLT     D13607 D13634  ; 查詢配方內容板材尺寸寬度設定 / 進料板寬(FLT)
      E/      D13634 E10 ZR2165  ; 進料板寬(FLT)
      FLT     D13608 D13636
      E/      D13636 E10 ZR2167
      FLT     D13609 D13638
      E/      D13638 E10 ZR2169
      FLT     D13610 D13640
      E/      D13640 E10 ZR2171
      FLT     D13611 D13642
      E/      D13642 E10 ZR2173
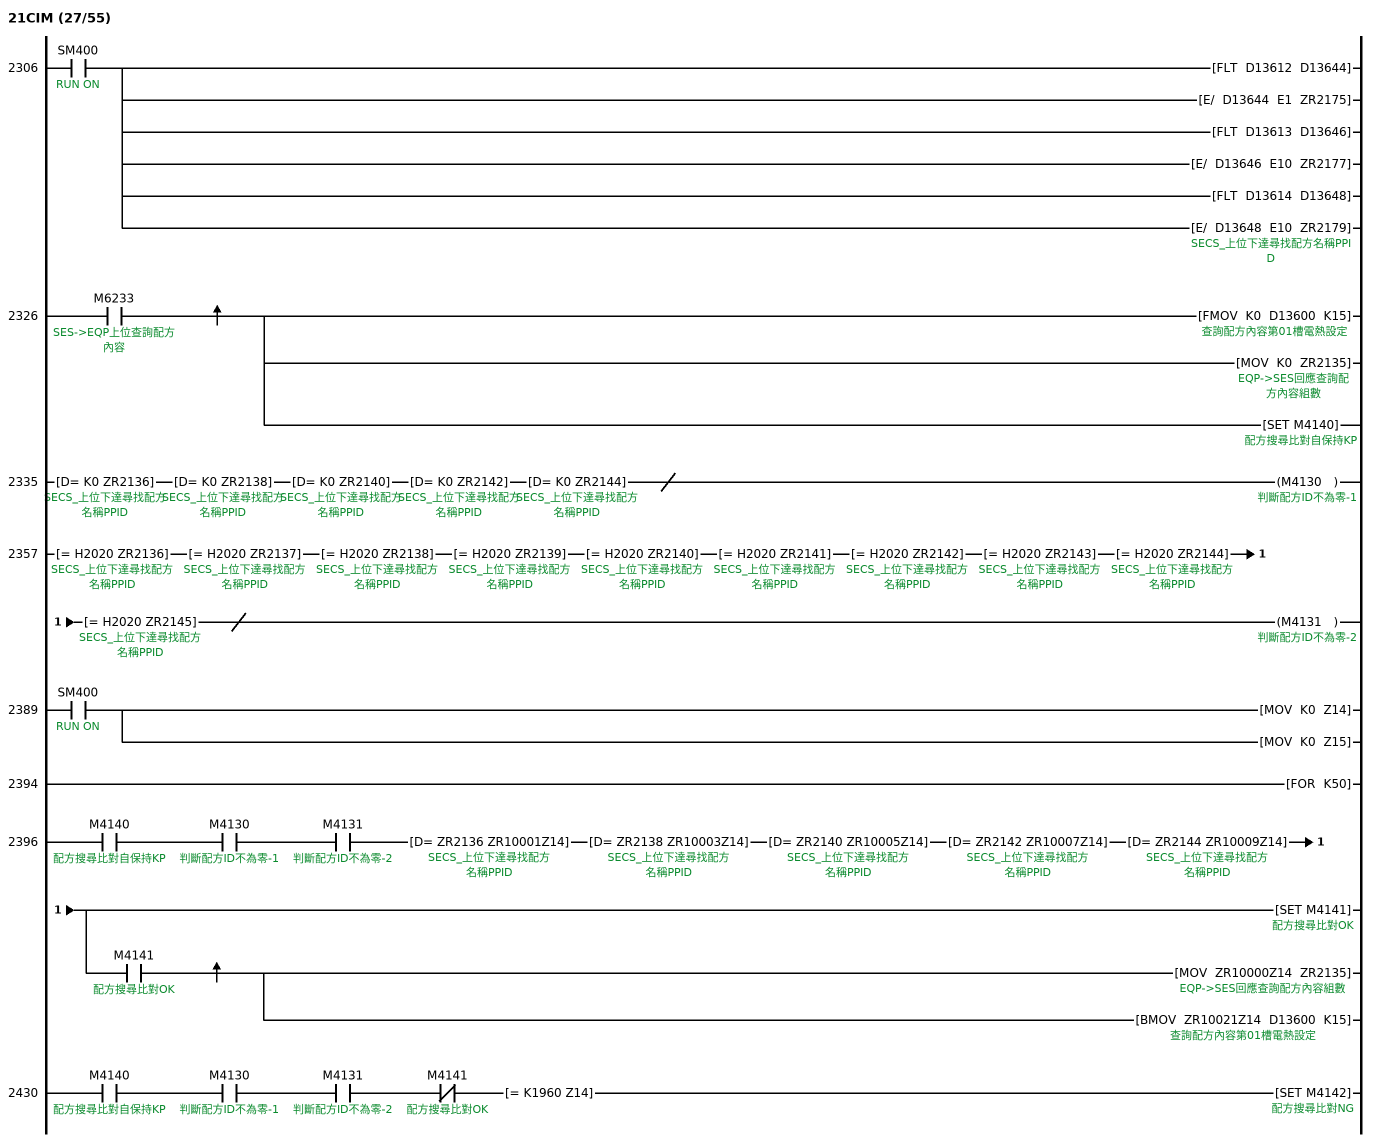
2306  LD      SM400  ; RUN ON
      FLT     D13612 D13644
      E/      D13644 E1 ZR2175
      FLT     D13613 D13646
      E/      D13646 E10 ZR2177
      FLT     D13614 D13648
      E/      D13648 E10 ZR2179  ; SECS_上位下達尋找配方名稱PPID
2326  LD      M6233  ; SES->EQP上位查詢配方內容
      MEP
      FMOV    K0 D13600 K15
      MOV     K0 ZR2135  ; EQP->SES回應查詢配方內容組數
      SET     M4140  ; 配方搜尋比對自保持KP
2335  LDD=    K0 ZR2136  ; SECS_上位下達尋找配方名稱PPID
      ANDD=   K0 ZR2138  ; SECS_上位下達尋找配方名稱PPID
      ANDD=   K0 ZR2140  ; SECS_上位下達尋找配方名稱PPID
      ANDD=   K0 ZR2142  ; SECS_上位下達尋找配方名稱PPID
      ANDD=   K0 ZR2144  ; SECS_上位下達尋找配方名稱PPID
      INV
      OUT     M4130  ; 判斷配方ID不為零-1
2357  LD=     H2020 ZR2136  ; SECS_上位下達尋找配方名稱PPID
      AND=    H2020 ZR2137  ; SECS_上位下達尋找配方名稱PPID
      AND=    H2020 ZR2138  ; SECS_上位下達尋找配方名稱PPID
      AND=    H2020 ZR2139  ; SECS_上位下達尋找配方名稱PPID
      AND=    H2020 ZR2140  ; SECS_上位下達尋找配方名稱PPID
      AND=    H2020 ZR2141  ; SECS_上位下達尋找配方名稱PPID
      AND=    H2020 ZR2142  ; SECS_上位下達尋找配方名稱PPID
      AND=    H2020 ZR2143  ; SECS_上位下達尋找配方名稱PPID
      AND=    H2020 ZR2144  ; SECS_上位下達尋找配方名稱PPID
      AND=    H2020 ZR2145  ; SECS_上位下達尋找配方名稱PPID
      INV
      OUT     M4131  ; 判斷配方ID不為零-2
2389  LD      SM400  ; RUN ON
      MOV     K0 Z14
      MOV     K0 Z15
2394  FOR     K50
2396  LD      M4140  ; 配方搜尋比對自保持KP
      AND     M4130  ; 判斷配方ID不為零-1
      AND     M4131  ; 判斷配方ID不為零-2
      ANDD=   ZR2136 ZR10001Z14  ; SECS_上位下達尋找配方名稱PPID
      ANDD=   ZR2138 ZR10003Z14  ; SECS_上位下達尋找配方名稱PPID
      ANDD=   ZR2140 ZR10005Z14  ; SECS_上位下達尋找配方名稱PPID
      ANDD=   ZR2142 ZR10007Z14  ; SECS_上位下達尋找配方名稱PPID
      ANDD=   ZR2144 ZR10009Z14  ; SECS_上位下達尋找配方名稱PPID
      SET     M4141  ; 配方搜尋比對OK
      AND     M4141  ; 配方搜尋比對OK
      MEP
      MOV     ZR10000Z14 ZR2135
      BMOV    ZR10021Z14 D13600 K15
2430  LD      M4140  ; 配方搜尋比對自保持KP
      AND     M4130  ; 判斷配方ID不為零-1
      AND     M4131  ; 判斷配方ID不為零-2
      ANI     M4141  ; 配方搜尋比對OK
      AND=    K1960 Z14
      SET     M4142  ; 配方搜尋比對NG
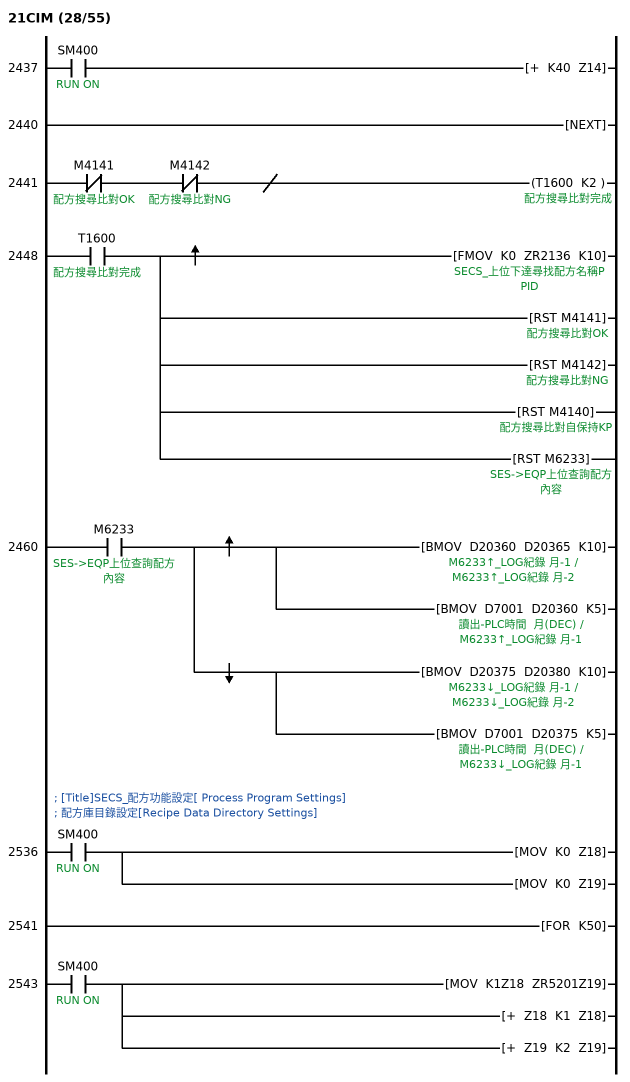
2437  LD      SM400  ; RUN ON
      +       K40 Z14
2440  NEXT
2441  LDI     M4141  ; 配方搜尋比對OK
      ANI     M4142  ; 配方搜尋比對NG
      INV
      OUT     T1600 K2  ; 配方搜尋比對完成
2448  LD      T1600  ; 配方搜尋比對完成
      MPS
      MEP
      FMOV    K0 ZR2136 K10
      MPP
      RST     M4141  ; 配方搜尋比對OK
      RST     M4142  ; 配方搜尋比對NG
      RST     M4140  ; 配方搜尋比對自保持KP
      RST     M6233  ; SES->EQP上位查詢配方內容
2460  LD      M6233  ; SES->EQP上位查詢配方內容
      MPS
      MEP
      BMOV    D20360 D20365 K10  ; M6233↑_LOG紀錄 月-1 / M6233↑_LOG紀錄 月-2
      BMOV    D7001 D20360 K5
      MPP
      MEF
      BMOV    D20375 D20380 K10  ; M6233↓_LOG紀錄 月-1 / M6233↓_LOG紀錄 月-2
      BMOV    D7001 D20375 K5
; [Title]SECS_配方功能設定[ Process Program Settings]
; 配方庫目錄設定[Recipe Data Directory Settings]
2536  LD      SM400  ; RUN ON
      MOV     K0 Z18
      MOV     K0 Z19
2541  FOR     K50
2543  LD      SM400  ; RUN ON
      MOV     K1Z18 ZR5201Z19
      +       Z18 K1 Z18
      +       Z19 K2 Z19
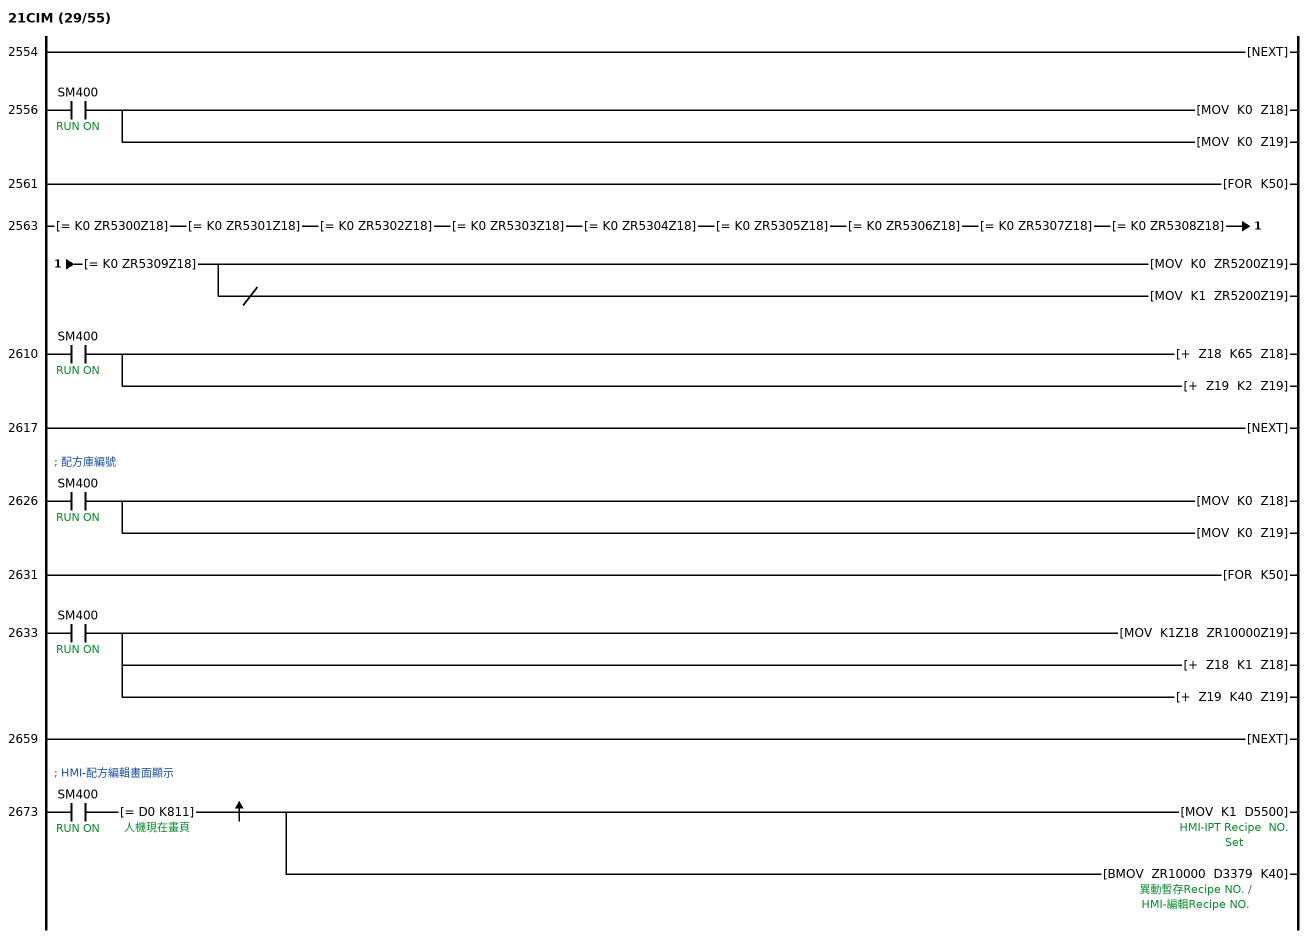
2554  NEXT
2556  LD      SM400  ; RUN ON
      MOV     K0 Z18
      MOV     K0 Z19
2561  FOR     K50
2563  LD=     K0 ZR5300Z18
      AND=    K0 ZR5301Z18
      AND=    K0 ZR5302Z18
      AND=    K0 ZR5303Z18
      AND=    K0 ZR5304Z18
      AND=    K0 ZR5305Z18
      AND=    K0 ZR5306Z18
      AND=    K0 ZR5307Z18
      AND=    K0 ZR5308Z18
      AND=    K0 ZR5309Z18
      MOV     K0 ZR5200Z19
      INV
      MOV     K1 ZR5200Z19
2610  LD      SM400  ; RUN ON
      +       Z18 K65 Z18
      +       Z19 K2 Z19
2617  NEXT
; 配方庫編號
2626  LD      SM400  ; RUN ON
      MOV     K0 Z18
      MOV     K0 Z19
2631  FOR     K50
2633  LD      SM400  ; RUN ON
      MOV     K1Z18 ZR10000Z19
        [note] 寫入配方參數Recipe NO.編號
      +       Z18 K1 Z18
      +       Z19 K40 Z19
2659  NEXT
; HMI-配方編輯畫面顯示
2673  LD      SM400  ; RUN ON
      AND=    D0 K811  ; 人機現在畫頁
      MEP
      MOV     K1 D5500  ; HMI-IPT Recipe  NO. Set
      BMOV    ZR10000 D3379 K40  ; 異動暫存Recipe NO. / HMI-編輯Recipe NO.
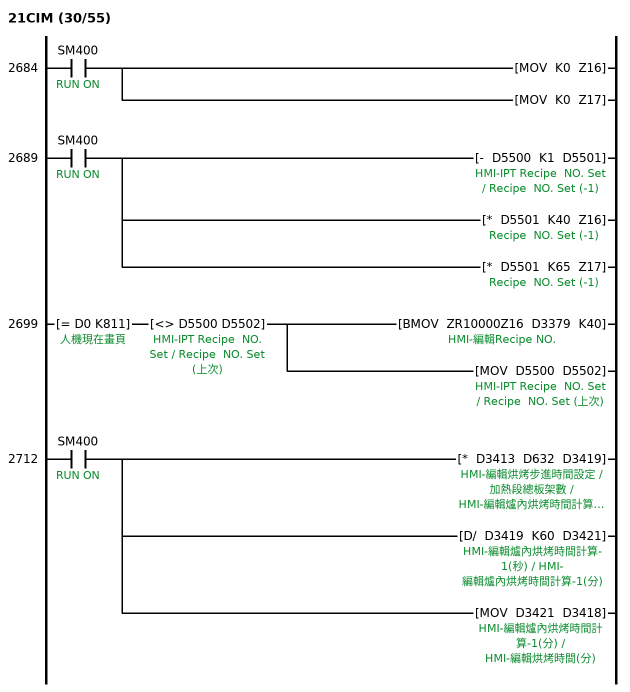
2684  LD      SM400  ; RUN ON
      MOV     K0 Z16
      MOV     K0 Z17
2689  LD      SM400  ; RUN ON
      -       D5500 K1 D5501  ; Recipe  NO. Set (-1)
      *       D5501 K40 Z16
      *       D5501 K65 Z17
2699  LD=     D0 K811  ; 人機現在畫頁
      AND<>   D5500 D5502  ; HMI-IPT Recipe  NO. Set / Recipe  NO. Set (上次)
      BMOV    ZR10000Z16 D3379 K40
      MOV     D5500 D5502
2712  LD      SM400  ; RUN ON
      *       D3413 D632 D3419  ; HMI-編輯烘烤步進時間設定 / 加熱段總板架數 / HMI-編輯爐內烘烤時間計算-1(秒)
        [note] 顯示輸入的秒數換算烘烤時間設定
      D/      D3419 K60 D3421  ; HMI-編輯爐內烘烤時間計算-1(分)
      MOV     D3421 D3418  ; HMI-編輯烘烤時間(分)
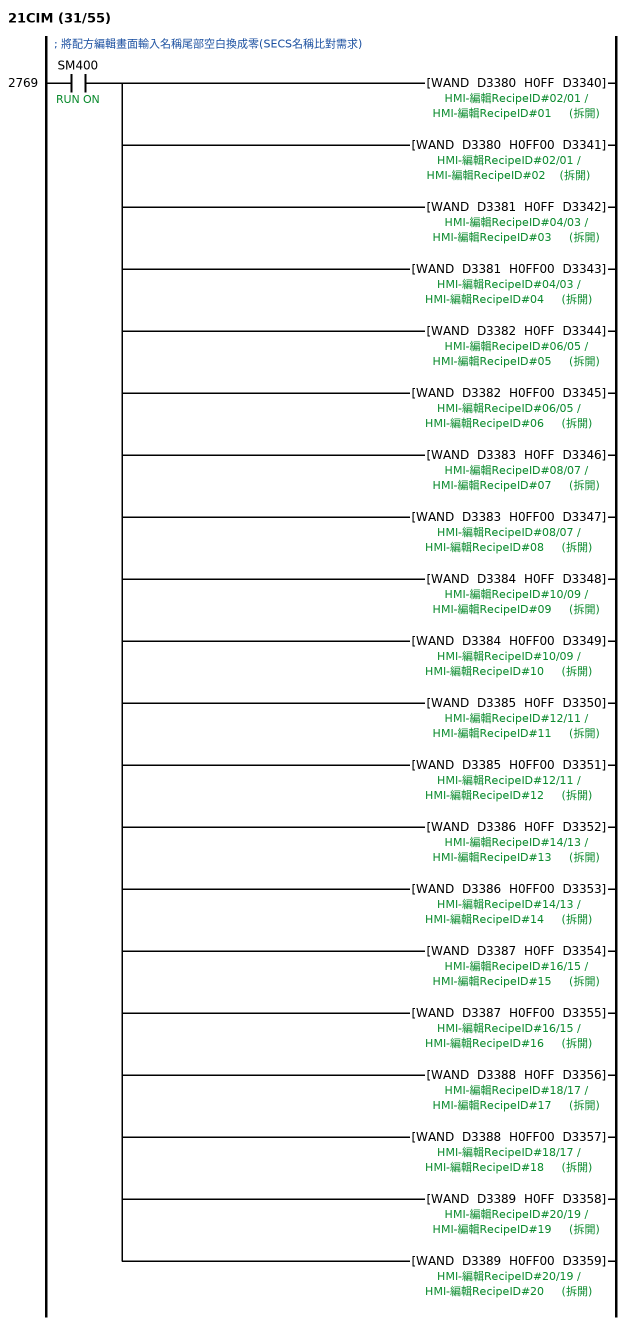
; 將配方編輯畫面輸入名稱尾部空白換成零(SECS名稱比對需求)
2769  LD      SM400  ; RUN ON
      WAND    D3380 H0FF D3340  ; HMI-編輯RecipeID#02/01 / HMI-編輯RecipeID#01     (拆開)
      WAND    D3380 H0FF00 D3341  ; HMI-編輯RecipeID#02    (拆開)
      WAND    D3381 H0FF D3342  ; HMI-編輯RecipeID#04/03 / HMI-編輯RecipeID#03     (拆開)
      WAND    D3381 H0FF00 D3343  ; HMI-編輯RecipeID#04     (拆開)
      WAND    D3382 H0FF D3344  ; HMI-編輯RecipeID#06/05 / HMI-編輯RecipeID#05     (拆開)
      WAND    D3382 H0FF00 D3345  ; HMI-編輯RecipeID#06     (拆開)
      WAND    D3383 H0FF D3346  ; HMI-編輯RecipeID#08/07 / HMI-編輯RecipeID#07     (拆開)
      WAND    D3383 H0FF00 D3347  ; HMI-編輯RecipeID#08     (拆開)
      WAND    D3384 H0FF D3348  ; HMI-編輯RecipeID#10/09 / HMI-編輯RecipeID#09     (拆開)
      WAND    D3384 H0FF00 D3349  ; HMI-編輯RecipeID#10     (拆開)
      WAND    D3385 H0FF D3350  ; HMI-編輯RecipeID#12/11 / HMI-編輯RecipeID#11     (拆開)
      WAND    D3385 H0FF00 D3351  ; HMI-編輯RecipeID#12     (拆開)
      WAND    D3386 H0FF D3352  ; HMI-編輯RecipeID#14/13 / HMI-編輯RecipeID#13     (拆開)
      WAND    D3386 H0FF00 D3353  ; HMI-編輯RecipeID#14     (拆開)
      WAND    D3387 H0FF D3354  ; HMI-編輯RecipeID#16/15 / HMI-編輯RecipeID#15     (拆開)
      WAND    D3387 H0FF00 D3355  ; HMI-編輯RecipeID#16     (拆開)
      WAND    D3388 H0FF D3356  ; HMI-編輯RecipeID#18/17 / HMI-編輯RecipeID#17     (拆開)
      WAND    D3388 H0FF00 D3357  ; HMI-編輯RecipeID#18     (拆開)
      WAND    D3389 H0FF D3358  ; HMI-編輯RecipeID#20/19 / HMI-編輯RecipeID#19     (拆開)
      WAND    D3389 H0FF00 D3359  ; HMI-編輯RecipeID#20     (拆開)
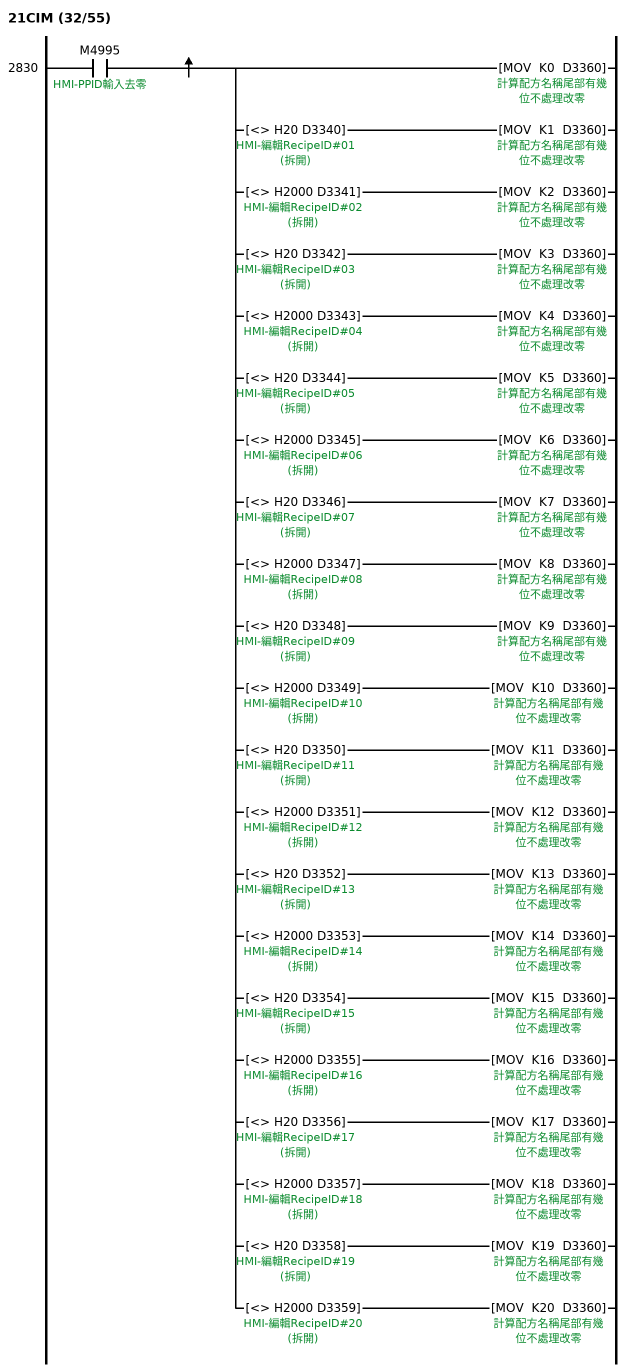
2830  LD      M4995  ; HMI-PPID輸入去零
      MEP
      MOV     K0 D3360  ; 計算配方名稱尾部有幾位不處理改零
      MPS
      AND<>   H20 D3340  ; HMI-編輯RecipeID#01     (拆開)
      MOV     K1 D3360
      MRD
      AND<>   H2000 D3341  ; HMI-編輯RecipeID#02    (拆開)
      MOV     K2 D3360
      MRD
      AND<>   H20 D3342  ; HMI-編輯RecipeID#03     (拆開)
      MOV     K3 D3360
      MRD
      AND<>   H2000 D3343  ; HMI-編輯RecipeID#04     (拆開)
      MOV     K4 D3360
      MRD
      AND<>   H20 D3344  ; HMI-編輯RecipeID#05     (拆開)
      MOV     K5 D3360
      MRD
      AND<>   H2000 D3345  ; HMI-編輯RecipeID#06     (拆開)
      MOV     K6 D3360
      MRD
      AND<>   H20 D3346  ; HMI-編輯RecipeID#07     (拆開)
      MOV     K7 D3360
      MRD
      AND<>   H2000 D3347  ; HMI-編輯RecipeID#08     (拆開)
      MOV     K8 D3360
      MRD
      AND<>   H20 D3348  ; HMI-編輯RecipeID#09     (拆開)
      MOV     K9 D3360
      MRD
      AND<>   H2000 D3349  ; HMI-編輯RecipeID#10     (拆開)
      MOV     K10 D3360
      MRD
      AND<>   H20 D3350  ; HMI-編輯RecipeID#11     (拆開)
      MOV     K11 D3360
      MRD
      AND<>   H2000 D3351  ; HMI-編輯RecipeID#12     (拆開)
      MOV     K12 D3360
      MRD
      AND<>   H20 D3352  ; HMI-編輯RecipeID#13     (拆開)
      MOV     K13 D3360
      MRD
      AND<>   H2000 D3353  ; HMI-編輯RecipeID#14     (拆開)
      MOV     K14 D3360
      MRD
      AND<>   H20 D3354  ; HMI-編輯RecipeID#15     (拆開)
      MOV     K15 D3360
      MRD
      AND<>   H2000 D3355  ; HMI-編輯RecipeID#16     (拆開)
      MOV     K16 D3360
      MRD
      AND<>   H20 D3356  ; HMI-編輯RecipeID#17     (拆開)
      MOV     K17 D3360
      MRD
      AND<>   H2000 D3357  ; HMI-編輯RecipeID#18     (拆開)
      MOV     K18 D3360
      MRD
      AND<>   H20 D3358  ; HMI-編輯RecipeID#19     (拆開)
      MOV     K19 D3360
      MPP
      AND<>   H2000 D3359  ; HMI-編輯RecipeID#20     (拆開)
      MOV     K20 D3360
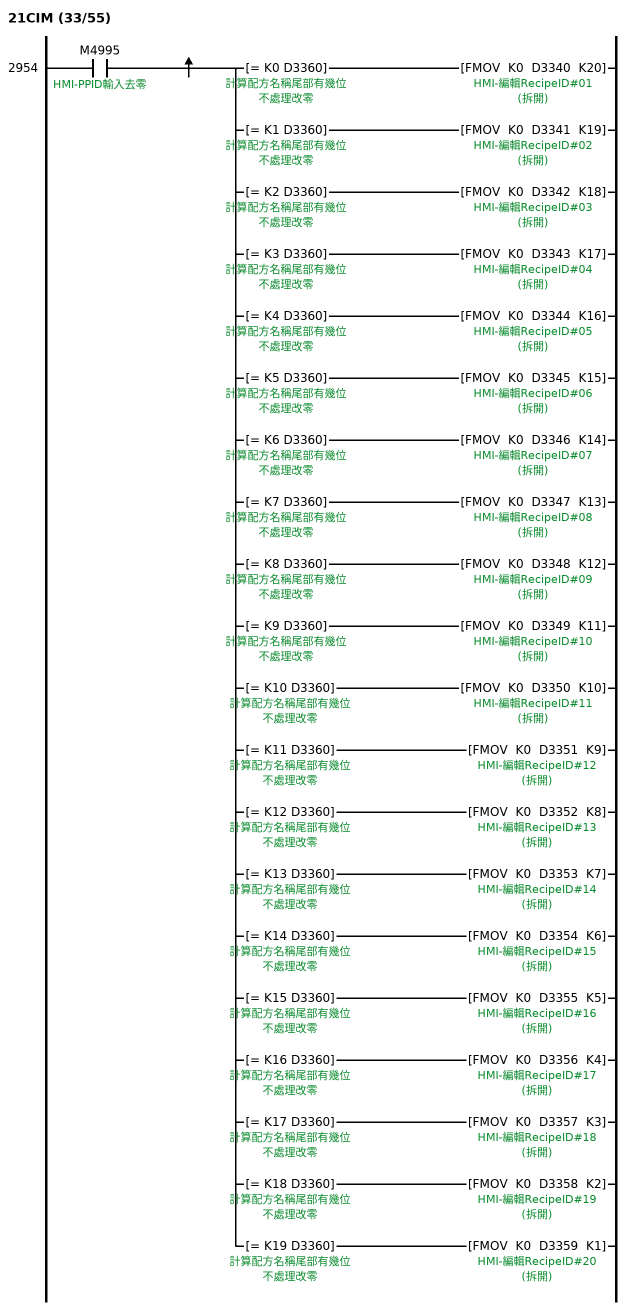
2954  LD      M4995  ; HMI-PPID輸入去零
      MEP
      MPS
      AND=    K0 D3360  ; 計算配方名稱尾部有幾位不處理改零
      FMOV    K0 D3340 K20
      MRD
      AND=    K1 D3360  ; 計算配方名稱尾部有幾位不處理改零
      FMOV    K0 D3341 K19
      MRD
      AND=    K2 D3360  ; 計算配方名稱尾部有幾位不處理改零
      FMOV    K0 D3342 K18
      MRD
      AND=    K3 D3360  ; 計算配方名稱尾部有幾位不處理改零
      FMOV    K0 D3343 K17
      MRD
      AND=    K4 D3360  ; 計算配方名稱尾部有幾位不處理改零
      FMOV    K0 D3344 K16
      MRD
      AND=    K5 D3360  ; 計算配方名稱尾部有幾位不處理改零
      FMOV    K0 D3345 K15
      MRD
      AND=    K6 D3360  ; 計算配方名稱尾部有幾位不處理改零
      FMOV    K0 D3346 K14
      MRD
      AND=    K7 D3360  ; 計算配方名稱尾部有幾位不處理改零
      FMOV    K0 D3347 K13
      MRD
      AND=    K8 D3360  ; 計算配方名稱尾部有幾位不處理改零
      FMOV    K0 D3348 K12
      MRD
      AND=    K9 D3360  ; 計算配方名稱尾部有幾位不處理改零
      FMOV    K0 D3349 K11
      MRD
      AND=    K10 D3360  ; 計算配方名稱尾部有幾位不處理改零
      FMOV    K0 D3350 K10
      MRD
      AND=    K11 D3360  ; 計算配方名稱尾部有幾位不處理改零
      FMOV    K0 D3351 K9
      MRD
      AND=    K12 D3360  ; 計算配方名稱尾部有幾位不處理改零
      FMOV    K0 D3352 K8
      MRD
      AND=    K13 D3360  ; 計算配方名稱尾部有幾位不處理改零
      FMOV    K0 D3353 K7
      MRD
      AND=    K14 D3360  ; 計算配方名稱尾部有幾位不處理改零
      FMOV    K0 D3354 K6
      MRD
      AND=    K15 D3360  ; 計算配方名稱尾部有幾位不處理改零
      FMOV    K0 D3355 K5
      MRD
      AND=    K16 D3360  ; 計算配方名稱尾部有幾位不處理改零
      FMOV    K0 D3356 K4
      MRD
      AND=    K17 D3360  ; 計算配方名稱尾部有幾位不處理改零
      FMOV    K0 D3357 K3
      MRD
      AND=    K18 D3360  ; 計算配方名稱尾部有幾位不處理改零
      FMOV    K0 D3358 K2
      MPP
      AND=    K19 D3360  ; 計算配方名稱尾部有幾位不處理改零
      FMOV    K0 D3359 K1
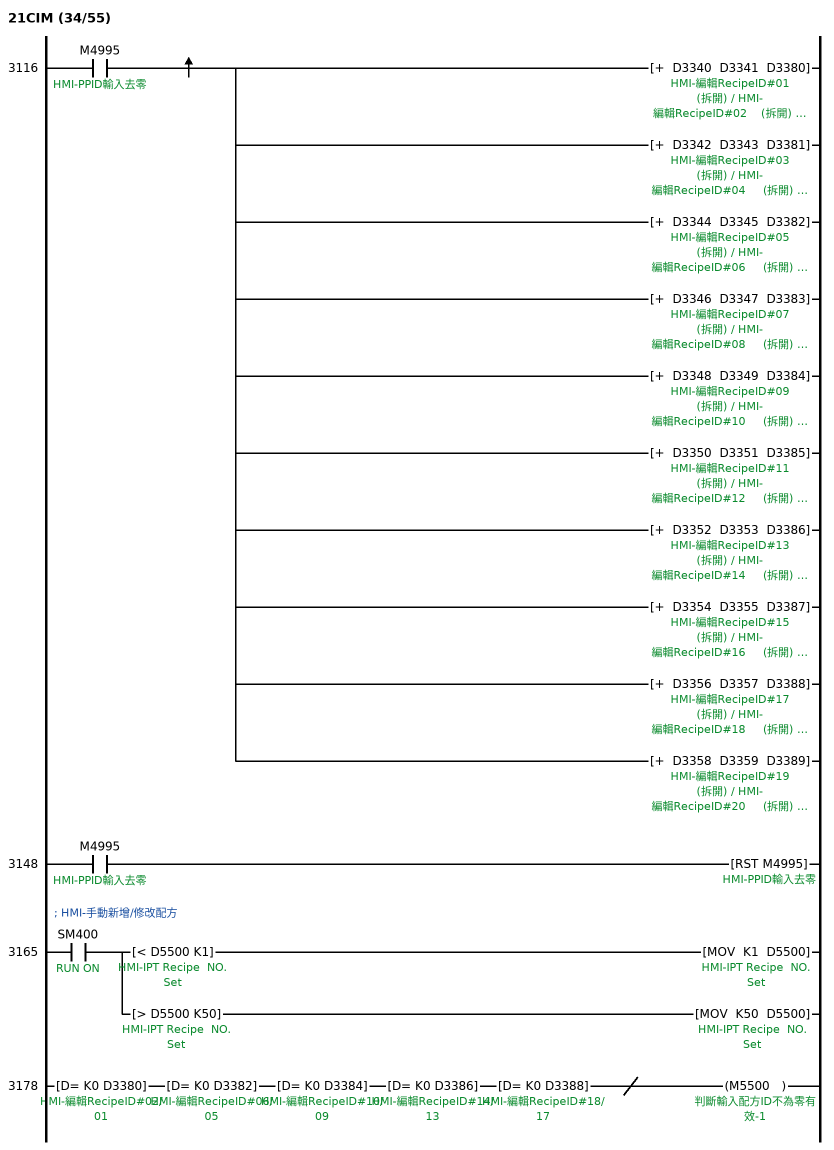
3116  LD      M4995  ; HMI-PPID輸入去零
      MEP
      +       D3340 D3341 D3380
      +       D3342 D3343 D3381
      +       D3344 D3345 D3382
      +       D3346 D3347 D3383
      +       D3348 D3349 D3384
      +       D3350 D3351 D3385
      +       D3352 D3353 D3386
      +       D3354 D3355 D3387
      +       D3356 D3357 D3388
      +       D3358 D3359 D3389
3148  LD      M4995  ; HMI-PPID輸入去零
      RST     M4995  ; HMI-PPID輸入去零
; HMI-手動新增/修改配方
3165  LD      SM400  ; RUN ON
      MPS
      AND<    D5500 K1  ; HMI-IPT Recipe  NO. Set
      MOV     K1 D5500
      MPP
      AND>    D5500 K50  ; HMI-IPT Recipe  NO. Set
      MOV     K50 D5500
3178  LDD=    K0 D3380  ; HMI-編輯RecipeID#02/01
      ANDD=   K0 D3382  ; HMI-編輯RecipeID#06/05
      ANDD=   K0 D3384  ; HMI-編輯RecipeID#10/09
      ANDD=   K0 D3386  ; HMI-編輯RecipeID#14/13
      ANDD=   K0 D3388  ; HMI-編輯RecipeID#18/17
      INV
      OUT     M5500  ; 判斷輸入配方ID不為零有效-1
